	{attribute 'TcIecLibraryType'}
	{attribute 'external_name' := 'F_VN_ReadDataMatrixCode_GUID_2844DFEA_73D9_3166_383A_C70A652858C4'}
	(* Detect and interpret a data matrix code within the provided image. *)
	FUNCTION F_VN_ReadDataMatrixCode : HRESULT
	VAR_INPUT
		ipSrcImage	:	ITcVnImage;	(* Source image (USINT elements, 1 or 3 channels) *)
		ipDecodedData	:	REFERENCE TO ITcVnContainer;	(* Returns the decoded code (ContainerType_Vector_String_SINT) *)
		hrPrev	:	HRESULT;	(* HRESULT indicating the result of previous operations (If SUCCEEDED(hrPrev) equals false, no operation is executed.) *)
	END_VAR

END_FUNCTION

// Functions/Code Reading/F_VN_ReadDataMatrixCodeExp

	{attribute 'TcIecLibraryType'}
	{attribute 'external_name' := 'F_VN_ReadDataMatrixCodeExp_GUID_B61F2F2C_5B12_3E0F_1052_05187753987C'}
	(* Detect and interpret a data matrix code within the provided image. *)
	FUNCTION F_VN_ReadDataMatrixCodeExp : HRESULT
	VAR_INPUT
		ipSrcImage	:	ITcVnImage;	(* Source image (USINT elements, 1 or 3 channels) *)
		ipDecodedData	:	REFERENCE TO ITcVnContainer;	(* Returns the decoded code (ContainerType_Vector_String_SINT) *)
		ipContours	:	REFERENCE TO ITcVnContainer;	(* Returns the code positions as contours (ContainerType_Vector_Vector_TcVnPoint2_DINT) *)
		nCodeNumber	:	DINT;	(* Number of data matrix codes that should be detected within the provided image. (If set to -1, it is tried to detect all data matrix codes.) *)
		eSearchStrategy	:	UDINT;	(* Used search strategy (ETcVn2dCodeSearchStrategy) *)
		hrPrev	:	HRESULT;	(* HRESULT indicating the result of previous operations (If SUCCEEDED(hrPrev) equals false, no operation is executed.) *)
	END_VAR

END_FUNCTION

// Functions/Code Reading/F_VN_ReadPharmaCode

	{attribute 'TcIecLibraryType'}
	{attribute 'external_name' := 'F_VN_ReadPharmaCode_GUID_7AF29CDE_1633_3CD4_1E1F_1FA9D1B23190'}
	(* Detect and interpret a pharma code within the provided image.
				Can be canceled by Watchdog. *)
	FUNCTION F_VN_ReadPharmaCode : HRESULT
	VAR_INPUT
		ipSrcImage	:	ITcVnImage;	(* Source image (1 channel (all element types) or 3 channel with elements of type TCVN_ET_USINT, TCVN_ET_UINT or TCVN_ET_REAL (3 channel input is expected to be RGB and internally converted to Gray)) *)
		ipDecodedData	:	REFERENCE TO ITcVnContainer;	(* Returns the decoded code (ContainerType_Vector_String_SINT) *)
		hrPrev	:	HRESULT;	(* HRESULT indicating the result of previous operations (If SUCCEEDED(hrPrev) equals false, no operation is executed.) *)
	END_VAR

END_FUNCTION

// Functions/Code Reading/F_VN_ReadPharmaCodeExp

	{attribute 'TcIecLibraryType'}
	{attribute 'external_name' := 'F_VN_ReadPharmaCodeExp_GUID_7FECB9FD_CF47_3BD7_11A2_73B8C61437DB'}
	(* Detect and interpret a pharma code within the provided image.
				Can be canceled by Watchdog. *)
	FUNCTION F_VN_ReadPharmaCodeExp : HRESULT
	VAR_INPUT
		ipSrcImage	:	ITcVnImage;	(* Source image (1 channel (all element types) or 3 channel with elements of type TCVN_ET_USINT, TCVN_ET_UINT or TCVN_ET_REAL (3 channel input is expected to be RGB and internally converted to Gray)) *)
		ipDecodedData	:	REFERENCE TO ITcVnContainer;	(* Returns the decoded code (ContainerType_Vector_String_SINT) *)
		ipContours	:	REFERENCE TO ITcVnContainer;	(* Returns the code positions as contours (ContainerType_Vector_Vector_TcVnPoint2_DINT) *)
		nCodeNumber	:	DINT;	(* Number of pharma codes that should be detected within the provided image (currently only 1 supported). *)
		nMinBarNumber	:	INT;	(* Minimal number of (dark) bars that codes must have. *)
		hrPrev	:	HRESULT;	(* HRESULT indicating the result of previous operations (If SUCCEEDED(hrPrev) equals false, no operation is executed.) *)
	END_VAR

END_FUNCTION

// Functions/Code Reading/F_VN_ReadQRCode

	{attribute 'TcIecLibraryType'}
	{attribute 'external_name' := 'F_VN_ReadQRCode_GUID_FDADFE2B_041B_3714_35C5_CCC4D2EB5C52'}
	(* Detect and interpret a QR code within the provided image.
          Can be canceled by Watchdog. *)
	FUNCTION F_VN_ReadQRCode : HRESULT
	VAR_INPUT
		ipSrcImage	:	ITcVnImage;	(* Source image (USINT elements, 1 channel or 3 channel (3 channel input is expected to be RGB and internally converted to Gray)) *)
		ipDecodedData	:	REFERENCE TO ITcVnContainer;	(* Returns the decoded code (ContainerType_Vector_String_SINT) *)
		hrPrev	:	HRESULT;	(* HRESULT indicating the result of previous operations (If SUCCEEDED(hrPrev) equals false, no operation is executed.) *)
	END_VAR

END_FUNCTION

// Functions/Code Reading/F_VN_ReadQRCodeExp

	{attribute 'TcIecLibraryType'}
	{attribute 'external_name' := 'F_VN_ReadQRCodeExp_GUID_701D058E_193D_312D_3EA8_971256078500'}
	(* Detect and interpret a QR code within the provided image.
          Can be canceled by Watchdog. *)
	FUNCTION F_VN_ReadQRCodeExp : HRESULT
	VAR_INPUT
		ipSrcImage	:	ITcVnImage;	(* Source image (USINT elements, 1 channel or 3 channel (3 channel input is expected to be RGB and internally converted to Gray)) *)
		ipDecodedData	:	REFERENCE TO ITcVnContainer;	(* Returns the decoded code (ContainerType_Vector_String_SINT) *)
		ipContours	:	REFERENCE TO ITcVnContainer;	(* Returns the code positions as contours (ContainerType_Vector_Vector_TcVnPoint2_DINT) *)
		nCodeNumber	:	DINT;	(* Number of QR codes that should be detected within the provided image (currently only 1 supported). *)
		eSearchStrategy	:	UDINT;	(* Used search strategy (ETcVn2dCodeSearchStrategy) *)
		hrPrev	:	HRESULT;	(* HRESULT indicating the result of previous operations (If SUCCEEDED(hrPrev) equals false, no operation is executed.) *)
	END_VAR

END_FUNCTION

// Functions/Algebraic Container Operations/F_VN_AddToContainerElements/F_VN_AddToContainerElements_DINT

	{attribute 'TcIecLibraryType'}
	{attribute 'external_name' := 'F_VN_AddToContainerElements_DINT_GUID_5B932B1D_0AB0_3885_2F50_15772C7465B6'}
	(* Add a value to each container element. *)
	FUNCTION F_VN_AddToContainerElements_DINT : HRESULT
	VAR_INPUT
		nValue	:	DINT;	(* Value *)
		ipContainer	:	ITcVnContainer;	(* Container with DINT elements *)
		hrPrev	:	HRESULT;	(* HRESULT indicating the result of previous operations (If SUCCEEDED(hrPrev) equals false, no operation is executed.) *)
	END_VAR

END_FUNCTION

// Functions/Algebraic Container Operations/F_VN_AddToContainerElements/F_VN_AddToContainerElements_INT

	{attribute 'TcIecLibraryType'}
	{attribute 'external_name' := 'F_VN_AddToContainerElements_INT_GUID_8666D2A8_02E9_3A45_051D_A4854190DF10'}
	(* Add a value to each container element. *)
	FUNCTION F_VN_AddToContainerElements_INT : HRESULT
	VAR_INPUT
		nValue	:	INT;	(* Value *)
		ipContainer	:	ITcVnContainer;	(* Container with INT elements *)
		hrPrev	:	HRESULT;	(* HRESULT indicating the result of previous operations (If SUCCEEDED(hrPrev) equals false, no operation is executed.) *)
	END_VAR

END_FUNCTION

// Functions/Algebraic Container Operations/F_VN_AddToContainerElements/F_VN_AddToContainerElements_LREAL

	{attribute 'TcIecLibraryType'}
	{attribute 'external_name' := 'F_VN_AddToContainerElements_LREAL_GUID_E41AE159_0A04_3EFE_16AB_C8BFD4EDC43A'}
	(* Add a value to each container element. *)
	FUNCTION F_VN_AddToContainerElements_LREAL : HRESULT
	VAR_INPUT
		fValue	:	LREAL;	(* Value *)
		ipContainer	:	ITcVnContainer;	(* Container with LREAL elements *)
		hrPrev	:	HRESULT;	(* HRESULT indicating the result of previous operations (If SUCCEEDED(hrPrev) equals false, no operation is executed.) *)
	END_VAR

END_FUNCTION

// Functions/Algebraic Container Operations/F_VN_AddToContainerElements/F_VN_AddToContainerElements_REAL

	{attribute 'TcIecLibraryType'}
	{attribute 'external_name' := 'F_VN_AddToContainerElements_REAL_GUID_692D4EAD_61C5_34E3_07CE_2D6EFBC619FC'}
	(* Add a value to each container element. *)
	FUNCTION F_VN_AddToContainerElements_REAL : HRESULT
	VAR_INPUT
		fValue	:	REAL;	(* Value *)
		ipContainer	:	ITcVnContainer;	(* Container with REAL elements *)
		hrPrev	:	HRESULT;	(* HRESULT indicating the result of previous operations (If SUCCEEDED(hrPrev) equals false, no operation is executed.) *)
	END_VAR

END_FUNCTION

// Functions/Algebraic Container Operations/F_VN_AddToContainerElements/F_VN_AddToContainerElements_SINT

	{attribute 'TcIecLibraryType'}
	{attribute 'external_name' := 'F_VN_AddToContainerElements_SINT_GUID_226FCB6F_5B19_30F7_05FC_4AEA7FD84914'}
	(* Add a value to each container element. *)
	FUNCTION F_VN_AddToContainerElements_SINT : HRESULT
	VAR_INPUT
		nValue	:	SINT;	(* Value *)
		ipContainer	:	ITcVnContainer;	(* Container with SINT elements *)
		hrPrev	:	HRESULT;	(* HRESULT indicating the result of previous operations (If SUCCEEDED(hrPrev) equals false, no operation is executed.) *)
	END_VAR

END_FUNCTION

// Functions/Algebraic Container Operations/F_VN_AddToContainerElements/F_VN_AddToContainerElements_TcVnKeyPoint

	{attribute 'TcIecLibraryType'}
	{attribute 'external_name' := 'F_VN_AddToContainerElements_TcVnKeyPoint_GUID_3B5F4B12_691D_304E_2813_D0B80607BE3C'}
	(* Add a value to each container element. *)
	FUNCTION F_VN_AddToContainerElements_TcVnKeyPoint : HRESULT
	VAR_INPUT
		stValue	:	REFERENCE TO TcVnKeyPoint;	(* Value *)
		ipContainer	:	ITcVnContainer;	(* Container with TcVnKeyPoint elements *)
		hrPrev	:	HRESULT;	(* HRESULT indicating the result of previous operations (If SUCCEEDED(hrPrev) equals false, no operation is executed.) *)
	END_VAR

END_FUNCTION

// Functions/Algebraic Container Operations/F_VN_AddToContainerElements/F_VN_AddToContainerElements_TcVnPoint2_DINT

	{attribute 'TcIecLibraryType'}
	{attribute 'external_name' := 'F_VN_AddToContainerElements_TcVnPoint2_DINT_GUID_01834351_EA53_3313_1ABA_CB9AAEF6914A'}
	(* Add a value to each container element. *)
	FUNCTION F_VN_AddToContainerElements_TcVnPoint2_DINT : HRESULT
	VAR_INPUT
		aValue	:	REFERENCE TO TcVnPoint2_DINT;	(* Value *)
		ipContainer	:	ITcVnContainer;	(* Container with TcVnPoint2_DINT elements *)
		hrPrev	:	HRESULT;	(* HRESULT indicating the result of previous operations (If SUCCEEDED(hrPrev) equals false, no operation is executed.) *)
	END_VAR

END_FUNCTION

// Functions/Algebraic Container Operations/F_VN_AddToContainerElements/F_VN_AddToContainerElements_TcVnPoint2_LREAL

	{attribute 'TcIecLibraryType'}
	{attribute 'external_name' := 'F_VN_AddToContainerElements_TcVnPoint2_LREAL_GUID_43701B1D_E3A8_30C8_24E6_54A2EFDCAA91'}
	(* Add a value to each container element. *)
	FUNCTION F_VN_AddToContainerElements_TcVnPoint2_LREAL : HRESULT
	VAR_INPUT
		aValue	:	REFERENCE TO TcVnPoint2_LREAL;	(* Value *)
		ipContainer	:	ITcVnContainer;	(* Container with TcVnPoint2_LREAL elements *)
		hrPrev	:	HRESULT;	(* HRESULT indicating the result of previous operations (If SUCCEEDED(hrPrev) equals false, no operation is executed.) *)
	END_VAR

END_FUNCTION

// Functions/Algebraic Container Operations/F_VN_AddToContainerElements/F_VN_AddToContainerElements_TcVnPoint2_REAL

	{attribute 'TcIecLibraryType'}
	{attribute 'external_name' := 'F_VN_AddToContainerElements_TcVnPoint2_REAL_GUID_00905747_5375_3335_13FD_44D74374D245'}
	(* Add a value to each container element. *)
	FUNCTION F_VN_AddToContainerElements_TcVnPoint2_REAL : HRESULT
	VAR_INPUT
		aValue	:	REFERENCE TO TcVnPoint2_REAL;	(* Value *)
		ipContainer	:	ITcVnContainer;	(* Container with TcVnPoint2_REAL elements *)
		hrPrev	:	HRESULT;	(* HRESULT indicating the result of previous operations (If SUCCEEDED(hrPrev) equals false, no operation is executed.) *)
	END_VAR

END_FUNCTION

// Functions/Algebraic Container Operations/F_VN_AddToContainerElements/F_VN_AddToContainerElements_TcVnPoint3_LREAL

	{attribute 'TcIecLibraryType'}
	{attribute 'external_name' := 'F_VN_AddToContainerElements_TcVnPoint3_LREAL_GUID_839DAD36_31CD_3F38_311A_A016EB995C42'}
	(* Add a value to each container element. *)
	FUNCTION F_VN_AddToContainerElements_TcVnPoint3_LREAL : HRESULT
	VAR_INPUT
		aValue	:	REFERENCE TO TcVnPoint3_LREAL;	(* Value *)
		ipContainer	:	ITcVnContainer;	(* Container with TcVnPoint3_LREAL elements *)
		hrPrev	:	HRESULT;	(* HRESULT indicating the result of previous operations (If SUCCEEDED(hrPrev) equals false, no operation is executed.) *)
	END_VAR

END_FUNCTION

// Functions/Algebraic Container Operations/F_VN_AddToContainerElements/F_VN_AddToContainerElements_TcVnPoint3_REAL

	{attribute 'TcIecLibraryType'}
	{attribute 'external_name' := 'F_VN_AddToContainerElements_TcVnPoint3_REAL_GUID_7F806659_1D47_3D35_077C_CC3B8A9E940F'}
	(* Add a value to each container element. *)
	FUNCTION F_VN_AddToContainerElements_TcVnPoint3_REAL : HRESULT
	VAR_INPUT
		aValue	:	REFERENCE TO TcVnPoint3_REAL;	(* Value *)
		ipContainer	:	ITcVnContainer;	(* Container with TcVnPoint3_REAL elements *)
		hrPrev	:	HRESULT;	(* HRESULT indicating the result of previous operations (If SUCCEEDED(hrPrev) equals false, no operation is executed.) *)
	END_VAR

END_FUNCTION

// Functions/Algebraic Container Operations/F_VN_AddToContainerElements/F_VN_AddToContainerElements_TcVnRectangle_DINT

	{attribute 'TcIecLibraryType'}
	{attribute 'external_name' := 'F_VN_AddToContainerElements_TcVnRectangle_DINT_GUID_5752E0A5_0126_3CCC_0ED6_0FAF696F41AB'}
	(* Add a value to each container element. *)
	FUNCTION F_VN_AddToContainerElements_TcVnRectangle_DINT : HRESULT
	VAR_INPUT
		stValue	:	REFERENCE TO TcVnRectangle_DINT;	(* Value *)
		ipContainer	:	ITcVnContainer;	(* Container with TcVnRectangle_DINT elements *)
		hrPrev	:	HRESULT;	(* HRESULT indicating the result of previous operations (If SUCCEEDED(hrPrev) equals false, no operation is executed.) *)
	END_VAR

END_FUNCTION

// Functions/Algebraic Container Operations/F_VN_AddToContainerElements/F_VN_AddToContainerElements_TcVnVector2_DINT

	{attribute 'TcIecLibraryType'}
	{attribute 'external_name' := 'F_VN_AddToContainerElements_TcVnVector2_DINT_GUID_FD05239B_FA44_389E_2792_06A9AFDB811F'}
	(* Add a value to each container element. *)
	FUNCTION F_VN_AddToContainerElements_TcVnVector2_DINT : HRESULT
	VAR_INPUT
		aValue	:	REFERENCE TO TcVnVector2_DINT;	(* Value *)
		ipContainer	:	ITcVnContainer;	(* Container with TcVnVector2_DINT elements *)
		hrPrev	:	HRESULT;	(* HRESULT indicating the result of previous operations (If SUCCEEDED(hrPrev) equals false, no operation is executed.) *)
	END_VAR

END_FUNCTION

// Functions/Algebraic Container Operations/F_VN_AddToContainerElements/F_VN_AddToContainerElements_TcVnVector2_INT

	{attribute 'TcIecLibraryType'}
	{attribute 'external_name' := 'F_VN_AddToContainerElements_TcVnVector2_INT_GUID_5A7959AB_7E96_36FB_0F59_3CCB450F9AC2'}
	(* Add a value to each container element. *)
	FUNCTION F_VN_AddToContainerElements_TcVnVector2_INT : HRESULT
	VAR_INPUT
		aValue	:	REFERENCE TO TcVnVector2_INT;	(* Value *)
		ipContainer	:	ITcVnContainer;	(* Container with TcVnVector2_INT elements *)
		hrPrev	:	HRESULT;	(* HRESULT indicating the result of previous operations (If SUCCEEDED(hrPrev) equals false, no operation is executed.) *)
	END_VAR

END_FUNCTION

// Functions/Algebraic Container Operations/F_VN_AddToContainerElements/F_VN_AddToContainerElements_TcVnVector2_REAL

	{attribute 'TcIecLibraryType'}
	{attribute 'external_name' := 'F_VN_AddToContainerElements_TcVnVector2_REAL_GUID_1870524F_E8DF_343A_1F0A_A50A67E87D79'}
	(* Add a value to each container element. *)
	FUNCTION F_VN_AddToContainerElements_TcVnVector2_REAL : HRESULT
	VAR_INPUT
		aValue	:	REFERENCE TO TcVnVector2_REAL;	(* Value *)
		ipContainer	:	ITcVnContainer;	(* Container with TcVnVector2_REAL elements *)
		hrPrev	:	HRESULT;	(* HRESULT indicating the result of previous operations (If SUCCEEDED(hrPrev) equals false, no operation is executed.) *)
	END_VAR

END_FUNCTION

// Functions/Algebraic Container Operations/F_VN_AddToContainerElements/F_VN_AddToContainerElements_TcVnVector2_SINT

	{attribute 'TcIecLibraryType'}
	{attribute 'external_name' := 'F_VN_AddToContainerElements_TcVnVector2_SINT_GUID_BA86B28B_BD11_3A77_358B_D5CC18E5F5D5'}
	(* Add a value to each container element. *)
	FUNCTION F_VN_AddToContainerElements_TcVnVector2_SINT : HRESULT
	VAR_INPUT
		aValue	:	REFERENCE TO TcVnVector2_SINT;	(* Value *)
		ipContainer	:	ITcVnContainer;	(* Container with TcVnVector2_SINT elements *)
		hrPrev	:	HRESULT;	(* HRESULT indicating the result of previous operations (If SUCCEEDED(hrPrev) equals false, no operation is executed.) *)
	END_VAR

END_FUNCTION

// Functions/Algebraic Container Operations/F_VN_AddToContainerElements/F_VN_AddToContainerElements_TcVnVector2_UINT

	{attribute 'TcIecLibraryType'}
	{attribute 'external_name' := 'F_VN_AddToContainerElements_TcVnVector2_UINT_GUID_56354970_50D0_3E9A_1D26_63220324D232'}
	(* Add a value to each container element. *)
	FUNCTION F_VN_AddToContainerElements_TcVnVector2_UINT : HRESULT
	VAR_INPUT
		aValue	:	REFERENCE TO TcVnVector2_UINT;	(* Value *)
		ipContainer	:	ITcVnContainer;	(* Container with TcVnVector2_UINT elements *)
		hrPrev	:	HRESULT;	(* HRESULT indicating the result of previous operations (If SUCCEEDED(hrPrev) equals false, no operation is executed.) *)
	END_VAR

END_FUNCTION

// Functions/Algebraic Container Operations/F_VN_AddToContainerElements/F_VN_AddToContainerElements_TcVnVector2_USINT

	{attribute 'TcIecLibraryType'}
	{attribute 'external_name' := 'F_VN_AddToContainerElements_TcVnVector2_USINT_GUID_19808A36_72A8_3C12_006D_40846B9F72C1'}
	(* Add a value to each container element. *)
	FUNCTION F_VN_AddToContainerElements_TcVnVector2_USINT : HRESULT
	VAR_INPUT
		aValue	:	REFERENCE TO TcVnVector2_USINT;	(* Value *)
		ipContainer	:	ITcVnContainer;	(* Container with TcVnVector2_USINT elements *)
		hrPrev	:	HRESULT;	(* HRESULT indicating the result of previous operations (If SUCCEEDED(hrPrev) equals false, no operation is executed.) *)
	END_VAR

END_FUNCTION

// Functions/Algebraic Container Operations/F_VN_AddToContainerElements/F_VN_AddToContainerElements_TcVnVector3_INT

	{attribute 'TcIecLibraryType'}
	{attribute 'external_name' := 'F_VN_AddToContainerElements_TcVnVector3_INT_GUID_71DC03E7_7327_3F01_0329_49D058A39A31'}
	(* Add a value to each container element. *)
	FUNCTION F_VN_AddToContainerElements_TcVnVector3_INT : HRESULT
	VAR_INPUT
		aValue	:	REFERENCE TO TcVnVector3_INT;	(* Value *)
		ipContainer	:	ITcVnContainer;	(* Container with TcVnVector3_INT elements *)
		hrPrev	:	HRESULT;	(* HRESULT indicating the result of previous operations (If SUCCEEDED(hrPrev) equals false, no operation is executed.) *)
	END_VAR

END_FUNCTION

// Functions/Algebraic Container Operations/F_VN_AddToContainerElements/F_VN_AddToContainerElements_TcVnVector3_REAL

	{attribute 'TcIecLibraryType'}
	{attribute 'external_name' := 'F_VN_AddToContainerElements_TcVnVector3_REAL_GUID_07AE301A_FCD1_34F3_164A_C1B5204DF30F'}
	(* Add a value to each container element. *)
	FUNCTION F_VN_AddToContainerElements_TcVnVector3_REAL : HRESULT
	VAR_INPUT
		aValue	:	REFERENCE TO TcVnVector3_REAL;	(* Value *)
		ipContainer	:	ITcVnContainer;	(* Container with TcVnVector3_REAL elements *)
		hrPrev	:	HRESULT;	(* HRESULT indicating the result of previous operations (If SUCCEEDED(hrPrev) equals false, no operation is executed.) *)
	END_VAR

END_FUNCTION

// Functions/Algebraic Container Operations/F_VN_AddToContainerElements/F_VN_AddToContainerElements_TcVnVector3_SINT

	{attribute 'TcIecLibraryType'}
	{attribute 'external_name' := 'F_VN_AddToContainerElements_TcVnVector3_SINT_GUID_6B5F8825_61DA_34E0_2CA0_F82329D5E791'}
	(* Add a value to each container element. *)
	FUNCTION F_VN_AddToContainerElements_TcVnVector3_SINT : HRESULT
	VAR_INPUT
		aValue	:	REFERENCE TO TcVnVector3_SINT;	(* Value *)
		ipContainer	:	ITcVnContainer;	(* Container with TcVnVector3_SINT elements *)
		hrPrev	:	HRESULT;	(* HRESULT indicating the result of previous operations (If SUCCEEDED(hrPrev) equals false, no operation is executed.) *)
	END_VAR

END_FUNCTION

// Functions/Algebraic Container Operations/F_VN_AddToContainerElements/F_VN_AddToContainerElements_TcVnVector3_UINT

	{attribute 'TcIecLibraryType'}
	{attribute 'external_name' := 'F_VN_AddToContainerElements_TcVnVector3_UINT_GUID_C23A5AA0_44F7_3E02_1B8F_AF04E59BD1A4'}
	(* Add a value to each container element. *)
	FUNCTION F_VN_AddToContainerElements_TcVnVector3_UINT : HRESULT
	VAR_INPUT
		aValue	:	REFERENCE TO TcVnVector3_UINT;	(* Value *)
		ipContainer	:	ITcVnContainer;	(* Container with TcVnVector3_UINT elements *)
		hrPrev	:	HRESULT;	(* HRESULT indicating the result of previous operations (If SUCCEEDED(hrPrev) equals false, no operation is executed.) *)
	END_VAR

END_FUNCTION

// Functions/Algebraic Container Operations/F_VN_AddToContainerElements/F_VN_AddToContainerElements_TcVnVector3_USINT

	{attribute 'TcIecLibraryType'}
	{attribute 'external_name' := 'F_VN_AddToContainerElements_TcVnVector3_USINT_GUID_D752658B_8056_3256_1C1B_709D22CABB66'}
	(* Add a value to each container element. *)
	FUNCTION F_VN_AddToContainerElements_TcVnVector3_USINT : HRESULT
	VAR_INPUT
		aValue	:	REFERENCE TO TcVnVector3_USINT;	(* Value *)
		ipContainer	:	ITcVnContainer;	(* Container with TcVnVector3_USINT elements *)
		hrPrev	:	HRESULT;	(* HRESULT indicating the result of previous operations (If SUCCEEDED(hrPrev) equals false, no operation is executed.) *)
	END_VAR

END_FUNCTION

// Functions/Algebraic Container Operations/F_VN_AddToContainerElements/F_VN_AddToContainerElements_TcVnVector4_DINT

	{attribute 'TcIecLibraryType'}
	{attribute 'external_name' := 'F_VN_AddToContainerElements_TcVnVector4_DINT_GUID_D742BE97_80DB_3CB5_027E_781E374D608F'}
	(* Add a value to each container element. *)
	FUNCTION F_VN_AddToContainerElements_TcVnVector4_DINT : HRESULT
	VAR_INPUT
		aValue	:	REFERENCE TO TcVnVector4_DINT;	(* Value *)
		ipContainer	:	ITcVnContainer;	(* Container with TcVnVector4_DINT elements *)
		hrPrev	:	HRESULT;	(* HRESULT indicating the result of previous operations (If SUCCEEDED(hrPrev) equals false, no operation is executed.) *)
	END_VAR

END_FUNCTION

// Functions/Algebraic Container Operations/F_VN_AddToContainerElements/F_VN_AddToContainerElements_TcVnVector4_INT

	{attribute 'TcIecLibraryType'}
	{attribute 'external_name' := 'F_VN_AddToContainerElements_TcVnVector4_INT_GUID_57836443_D91C_30AD_0584_7CCF6B06E1D4'}
	(* Add a value to each container element. *)
	FUNCTION F_VN_AddToContainerElements_TcVnVector4_INT : HRESULT
	VAR_INPUT
		aValue	:	REFERENCE TO TcVnVector4_INT;	(* Value *)
		ipContainer	:	ITcVnContainer;	(* Container with TcVnVector4_INT elements *)
		hrPrev	:	HRESULT;	(* HRESULT indicating the result of previous operations (If SUCCEEDED(hrPrev) equals false, no operation is executed.) *)
	END_VAR

END_FUNCTION

// Functions/Algebraic Container Operations/F_VN_AddToContainerElements/F_VN_AddToContainerElements_TcVnVector4_LREAL

	{attribute 'TcIecLibraryType'}
	{attribute 'external_name' := 'F_VN_AddToContainerElements_TcVnVector4_LREAL_GUID_360561FB_FBFC_3471_3F24_900DC5ABA6EC'}
	(* Add a value to each container element. *)
	FUNCTION F_VN_AddToContainerElements_TcVnVector4_LREAL : HRESULT
	VAR_INPUT
		aValue	:	REFERENCE TO TcVnVector4_LREAL;	(* Value *)
		ipContainer	:	ITcVnContainer;	(* Container with TcVnVector4_LREAL elements *)
		hrPrev	:	HRESULT;	(* HRESULT indicating the result of previous operations (If SUCCEEDED(hrPrev) equals false, no operation is executed.) *)
	END_VAR

END_FUNCTION

// Functions/Algebraic Container Operations/F_VN_AddToContainerElements/F_VN_AddToContainerElements_TcVnVector4_SINT

	{attribute 'TcIecLibraryType'}
	{attribute 'external_name' := 'F_VN_AddToContainerElements_TcVnVector4_SINT_GUID_1820B1AC_0FF9_3EE1_38CE_685FDE758958'}
	(* Add a value to each container element. *)
	FUNCTION F_VN_AddToContainerElements_TcVnVector4_SINT : HRESULT
	VAR_INPUT
		aValue	:	REFERENCE TO TcVnVector4_SINT;	(* Value *)
		ipContainer	:	ITcVnContainer;	(* Container with TcVnVector4_SINT elements *)
		hrPrev	:	HRESULT;	(* HRESULT indicating the result of previous operations (If SUCCEEDED(hrPrev) equals false, no operation is executed.) *)
	END_VAR

END_FUNCTION

// Functions/Algebraic Container Operations/F_VN_AddToContainerElements/F_VN_AddToContainerElements_TcVnVector4_UINT

	{attribute 'TcIecLibraryType'}
	{attribute 'external_name' := 'F_VN_AddToContainerElements_TcVnVector4_UINT_GUID_5187AFB3_19BE_3EE8_32AD_0FFCFCC25933'}
	(* Add a value to each container element. *)
	FUNCTION F_VN_AddToContainerElements_TcVnVector4_UINT : HRESULT
	VAR_INPUT
		aValue	:	REFERENCE TO TcVnVector4_UINT;	(* Value *)
		ipContainer	:	ITcVnContainer;	(* Container with TcVnVector4_UINT elements *)
		hrPrev	:	HRESULT;	(* HRESULT indicating the result of previous operations (If SUCCEEDED(hrPrev) equals false, no operation is executed.) *)
	END_VAR

END_FUNCTION

// Functions/Algebraic Container Operations/F_VN_AddToContainerElements/F_VN_AddToContainerElements_TcVnVector4_USINT

	{attribute 'TcIecLibraryType'}
	{attribute 'external_name' := 'F_VN_AddToContainerElements_TcVnVector4_USINT_GUID_77580D86_B358_375A_06A3_8BDBEA39CE74'}
	(* Add a value to each container element. *)
	FUNCTION F_VN_AddToContainerElements_TcVnVector4_USINT : HRESULT
	VAR_INPUT
		aValue	:	REFERENCE TO TcVnVector4_USINT;	(* Value *)
		ipContainer	:	ITcVnContainer;	(* Container with TcVnVector4_USINT elements *)
		hrPrev	:	HRESULT;	(* HRESULT indicating the result of previous operations (If SUCCEEDED(hrPrev) equals false, no operation is executed.) *)
	END_VAR

END_FUNCTION

// Functions/Algebraic Container Operations/F_VN_AddToContainerElements/F_VN_AddToContainerElements_UDINT

	{attribute 'TcIecLibraryType'}
	{attribute 'external_name' := 'F_VN_AddToContainerElements_UDINT_GUID_5ECD52C6_7D8F_3D13_28F8_D2F1CCB21427'}
	(* Add a value to each container element. *)
	FUNCTION F_VN_AddToContainerElements_UDINT : HRESULT
	VAR_INPUT
		nValue	:	UDINT;	(* Value *)
		ipContainer	:	ITcVnContainer;	(* Container with UDINT elements *)
		hrPrev	:	HRESULT;	(* HRESULT indicating the result of previous operations (If SUCCEEDED(hrPrev) equals false, no operation is executed.) *)
	END_VAR

END_FUNCTION

// Functions/Algebraic Container Operations/F_VN_AddToContainerElements/F_VN_AddToContainerElements_UINT

	{attribute 'TcIecLibraryType'}
	{attribute 'external_name' := 'F_VN_AddToContainerElements_UINT_GUID_AAC9CFC5_57F2_382F_1BD9_9DFEB6B09CFB'}
	(* Add a value to each container element. *)
	FUNCTION F_VN_AddToContainerElements_UINT : HRESULT
	VAR_INPUT
		nValue	:	UINT;	(* Value *)
		ipContainer	:	ITcVnContainer;	(* Container with UINT elements *)
		hrPrev	:	HRESULT;	(* HRESULT indicating the result of previous operations (If SUCCEEDED(hrPrev) equals false, no operation is executed.) *)
	END_VAR

END_FUNCTION

// Functions/Algebraic Container Operations/F_VN_AddToContainerElements/F_VN_AddToContainerElements_ULINT

	{attribute 'TcIecLibraryType'}
	{attribute 'external_name' := 'F_VN_AddToContainerElements_ULINT_GUID_85BFEBDA_E705_31D3_2B59_BA00C1290486'}
	(* Add a value to each container element. *)
	FUNCTION F_VN_AddToContainerElements_ULINT : HRESULT
	VAR_INPUT
		nValue	:	ULINT;	(* Value *)
		ipContainer	:	ITcVnContainer;	(* Container with ULINT elements *)
		hrPrev	:	HRESULT;	(* HRESULT indicating the result of previous operations (If SUCCEEDED(hrPrev) equals false, no operation is executed.) *)
	END_VAR

END_FUNCTION

// Functions/Algebraic Container Operations/F_VN_AddToContainerElements/F_VN_AddToContainerElements_USINT

	{attribute 'TcIecLibraryType'}
	{attribute 'external_name' := 'F_VN_AddToContainerElements_USINT_GUID_5BF3EAE4_887F_3F25_01F9_F187751B7D61'}
	(* Add a value to each container element. *)
	FUNCTION F_VN_AddToContainerElements_USINT : HRESULT
	VAR_INPUT
		nValue	:	USINT;	(* Value *)
		ipContainer	:	ITcVnContainer;	(* Container with USINT elements *)
		hrPrev	:	HRESULT;	(* HRESULT indicating the result of previous operations (If SUCCEEDED(hrPrev) equals false, no operation is executed.) *)
	END_VAR

END_FUNCTION

// Functions/Image Analysis/Object Detection/F_VN_AdjustActiveContour

	{attribute 'TcIecLibraryType'}
	{attribute 'external_name' := 'F_VN_AdjustActiveContour_GUID_E8A83B8A_FFAF_376E_0EAC_1914E2C30A5B'}
	(* Adjust active contour (snake) in order to minimize its cummulative (internal and external) energy. *)
	FUNCTION F_VN_AdjustActiveContour : HRESULT
	VAR_INPUT
		ipImage	:	ITcVnImage;	(* Source image (1 channel, USINT elements) *)
		ipActiveContour	:	ITcVnContainer;	(* Initial contour, which will be adjusted *)
		fAlpha	:	REAL;	(* Continuity energy coefficient *)
		fBeta	:	REAL;	(* Curvature energy coefficient *)
		fGamma	:	REAL;	(* Image energy coefficient *)
		nWindowWidth	:	UDINT;	(* Windows width (3, 5, 7, ...) *)
		nWindowHeight	:	UDINT;	(* Windows height (3, 5, 7, ...) *)
		nMaxIterations	:	UDINT;	(* Maximum iterations *)
		bUseGradient	:	BOOL;	(* If true, the gradient magnitude is used as image energy (otherwise: pixel intensity) *)
		hrPrev	:	HRESULT;	(* HRESULT indicating the result of previous operations (If SUCCEEDED(hrPrev) equals false, no operation is executed.) *)
	END_VAR

END_FUNCTION

// Functions/Image Analysis/Object Detection/F_VN_DetectBlobs

	{attribute 'TcIecLibraryType'}
	{attribute 'external_name' := 'F_VN_DetectBlobs_GUID_D96B8C6D_95DC_37E7_33AE_CFA61E2C6332'}
	(* Detects blob-contours. Applies a threshold, a contour search and offers several options for filtering the found contours. Provides easy setup for multiple thresholds and combination of results. *)
	FUNCTION F_VN_DetectBlobs : HRESULT
	VAR_INPUT
		ipSrcImage	:	ITcVnImage;	(* Source image (USINT or REAL, 1 channel or 3 channel (3 channel input is expected to be RGB and internally converted to Gray)) *)
		ipBlobContours	:	REFERENCE TO ITcVnContainer;	(* Returns a container which is filled with the found contours (ContainerType_Vector_Vector_TcVnPoint2_DINT; The elements of this container are single contours. Non-zero interface pointers are reused.) *)
		stParams	:	REFERENCE TO TcVnParamsBlobDetection;	(* Parameters to filter the detected contours. *)
		hrPrev	:	HRESULT;	(* HRESULT indicating the result of previous operations (If SUCCEEDED(hrPrev) equals false, no operation is executed.) *)
	END_VAR

END_FUNCTION

// Functions/Image Analysis/Object Detection/F_VN_DetectBlobsExp

	{attribute 'TcIecLibraryType'}
	{attribute 'external_name' := 'F_VN_DetectBlobsExp_GUID_FC112C44_43B7_3777_1919_1F0811271198'}
	(* Detects blob-contours. Applies a threshold, a contour search and offers several options for filtering the found contours. Provides easy setup for multiple thresholds and combination of results. (expert function) *)
	FUNCTION F_VN_DetectBlobsExp : HRESULT
	VAR_INPUT
		ipSrcImage	:	ITcVnImage;	(* Source image (USINT or REAL, 1 channel or 3 channel (3 channel input is expected to be RGB and internally converted to Gray)) *)
		ipBlobContours	:	REFERENCE TO ITcVnContainer;	(* Returns a container which is filled with the found contours (ContainerType_Vector_Vector_TcVnPoint2_DINT; The elements of this container are single contours. Non-zero interface pointers are reused.) *)
		stParams	:	REFERENCE TO TcVnParamsBlobDetection;	(* Parameters to filter the detected contours. *)
		aOffset	:	REFERENCE TO TcVnPoint;	(* Offset by which every contour point is shifted *)
		hrPrev	:	HRESULT;	(* HRESULT indicating the result of previous operations (If SUCCEEDED(hrPrev) equals false, no operation is executed.) *)
	END_VAR

END_FUNCTION

// Functions/Image Analysis/Object Detection/F_VN_FindContourHierarchyExp

	{attribute 'TcIecLibraryType'}
	{attribute 'external_name' := 'F_VN_FindContourHierarchyExp_GUID_9473BECE_526D_34AA_1C97_88FE3EFAE71A'}
	(* Search for object contours in a binary image and determine their hierarchical relationship. (expert function) *)
	FUNCTION F_VN_FindContourHierarchyExp : HRESULT
	VAR_INPUT
		ipSrcImage	:	ITcVnImage;	(* Source image (1 channel, binary) *)
		ipContours	:	REFERENCE TO ITcVnContainer;	(* Returns a container which is filled with the found contours (ContainerType_Vector_Vector_TcVnPoint2_DINT; The elements of this container are single contours. Non-zero interface pointers are reused.) *)
		ipHierarchy	:	REFERENCE TO ITcVnContainer;	(* Returns a container which is filled with information on the found contours' hierarchy (ContainerType_Vector_TcVnVector4_DINT; The elements of this container are four-dimensional vectors containing the 0-based indices of the next [0] and the previous contour [1] at the same level, the first child [2], and the parent [3]. Non-zero interface pointers are reused.) *)
		eRetrievalMode	:	ETcVnContourRetrievalMode;	(* Specifies which contours are retrieved and how their relationship is encoded *)
		eApproximationMethod	:	ETcVnContourApproximationMethod;	(* Contour encoding *)
		aOffset	:	REFERENCE TO TcVnPoint;	(* Offset by which every contour point is shifted *)
		hrPrev	:	HRESULT;	(* HRESULT indicating the result of previous operations (If SUCCEEDED(hrPrev) equals false, no operation is executed.) *)
	END_VAR

END_FUNCTION

// Functions/Image Analysis/Object Detection/F_VN_FindContours

	{attribute 'TcIecLibraryType'}
	{attribute 'external_name' := 'F_VN_FindContours_GUID_FCB893B9_E591_3799_2A0C_20BA26051DE9'}
	(* Search for object contours in a binary image. Returns only external contours. *)
	FUNCTION F_VN_FindContours : HRESULT
	VAR_INPUT
		ipSrcImage	:	ITcVnImage;	(* Source image (1 channel, binary) *)
		ipContours	:	REFERENCE TO ITcVnContainer;	(* Returns a container which is filled with the found contours (ContainerType_Vector_Vector_TcVnPoint2_DINT; The elements of this container are single contours. Non-zero interface pointers are reused.) *)
		hrPrev	:	HRESULT;	(* HRESULT indicating the result of previous operations (If SUCCEEDED(hrPrev) equals false, no operation is executed.) *)
	END_VAR

END_FUNCTION

// Functions/Image Analysis/Object Detection/F_VN_FindContoursExp

	{attribute 'TcIecLibraryType'}
	{attribute 'external_name' := 'F_VN_FindContoursExp_GUID_8CBA5025_8ECB_358F_0E17_DE22AB7A2587'}
	(* Search for object contours in a binary image. (expert function) *)
	FUNCTION F_VN_FindContoursExp : HRESULT
	VAR_INPUT
		ipSrcImage	:	ITcVnImage;	(* Source image (1 channel, binary) *)
		ipContours	:	REFERENCE TO ITcVnContainer;	(* Returns a container which is filled with the found contours (ContainerType_Vector_Vector_TcVnPoint2_DINT; The elements of this container are single contours. Non-zero interface pointers are reused.) *)
		eRetrievalMode	:	ETcVnContourRetrievalMode;	(* Specifies which contours are retrieved and how their relationship is encoded *)
		eApproximationMethod	:	ETcVnContourApproximationMethod;	(* Contour encoding *)
		aOffset	:	REFERENCE TO TcVnPoint;	(* Offset by which every contour point is shifted *)
		hrPrev	:	HRESULT;	(* HRESULT indicating the result of previous operations (If SUCCEEDED(hrPrev) equals false, no operation is executed.) *)
	END_VAR

END_FUNCTION

// Functions/Image Analysis/Object Detection/F_VN_HoughCircles

	{attribute 'TcIecLibraryType'}
	{attribute 'external_name' := 'F_VN_HoughCircles_GUID_C629D5C8_F15A_3685_3EE3_DABA5DA8EF57'}
	(* Search for circles using the Hough transform. *)
	FUNCTION F_VN_HoughCircles : HRESULT
	VAR_INPUT
		ipSrcImage	:	ITcVnImage;	(* Source image (USINT, 1 channel, gray-level) *)
		ipCircles	:	REFERENCE TO ITcVnContainer;	(* Returns a container which is filled with the found circles (ContainerType_Vector_TcVnVector3_REAL; Each container element contains the x coordinate of the circle center [0], the y coordinate of the circle center [1], and the radius [2], respectively. Non-zero interface pointers are reused.) *)
		fInvAccuRatio	:	LREAL;	(* Inverted ratio of the accumulator size in relation to the source image's size (must be > 0. A value of 2 means that the size is halved in both directions.) *)
		fMinDist	:	LREAL;	(* Smallest allowed distance of two circles (must be > 0) *)
		hrPrev	:	HRESULT;	(* HRESULT indicating the result of previous operations (If SUCCEEDED(hrPrev) equals false, no operation is executed.) *)
	END_VAR

END_FUNCTION

// Functions/Image Analysis/Object Detection/F_VN_HoughCirclesExp

	{attribute 'TcIecLibraryType'}
	{attribute 'external_name' := 'F_VN_HoughCirclesExp_GUID_F105B70A_1E4C_3D67_2153_0BAD535BB162'}
	(* Search for circles using the Hough transform. (expert function) *)
	FUNCTION F_VN_HoughCirclesExp : HRESULT
	VAR_INPUT
		ipSrcImage	:	ITcVnImage;	(* Source image (USINT, 1 channel, gray-level) *)
		ipCircles	:	REFERENCE TO ITcVnContainer;	(* Returns a container which is filled with the found circles (ContainerType_Vector_TcVnVector3_REAL; Each container element contains the x coordinate of the circle center [0], the y coordinate of the circle center [1], and the radius [2], respectively. Non-zero interface pointers are reused.) *)
		fInvAccuRatio	:	LREAL;	(* Inverted ratio of the accumulator size in relation to the source image's size (must be > 0. A value of 2 means that the size is halved in both directions.) *)
		fMinDist	:	LREAL;	(* Smallest allowed distance of two circles (must be > 0) *)
		eHoughMethod	:	ETcVnHoughMethod;	(* Hough method to use (GRADIENT or GRADIENT_ALT) *)
		fParam1	:	LREAL;	(* First method specific parameter (GRADIENT, GRADIENT_ALT: upper threshold for canny edge detection, which must be > 0) *)
		fParam2	:	LREAL;	(* Second method specific parameter (GRADIENT: accumulator threshold for detecting circle centers, which must be > 0. GRADIENT_ALT: required circle perfectness, which must be > 0 and < 1, 1 would be a perfect circle) *)
		nMinRadius	:	UDINT;	(* Minimum circle radius allowed *)
		nMaxRadius	:	UDINT;	(* Maximum circle radius allowed (if 0, the value is internally set to max(image rows, image columns)) *)
		hrPrev	:	HRESULT;	(* HRESULT indicating the result of previous operations (If SUCCEEDED(hrPrev) equals false, no operation is executed.) *)
	END_VAR

END_FUNCTION

// Functions/Image Analysis/Object Detection/F_VN_HoughLines

	{attribute 'TcIecLibraryType'}
	{attribute 'external_name' := 'F_VN_HoughLines_GUID_769839FF_1529_3A59_2422_8F8DC7D5C4E7'}
	(* Search for lines using the standard Hough transform. *)
	FUNCTION F_VN_HoughLines : HRESULT
	VAR_INPUT
		ipSrcImage	:	ITcVnImage;	(* Source image (USINT, 1 channel, binary, may be modified by the function) *)
		ipLines	:	REFERENCE TO ITcVnContainer;	(* Returns a container which is filled with the found lines (ContainerType_Vector_TcVnVector2_REAL; Each container element contains the distance from the origin [0] in pixels and the rotation angle [1] in radians, respectively. Non-zero interface pointers are reused.) *)
		fDistRes	:	LREAL;	(* Distance resolution of the accumulator (in pixels, must be > 0) *)
		fAngleRes	:	LREAL;	(* Angle resolution of the accumulator (in radians, must be > 0) *)
		nAccuThreshold	:	UDINT;	(* Accumulator threshold *)
		hrPrev	:	HRESULT;	(* HRESULT indicating the result of previous operations (If SUCCEEDED(hrPrev) equals false, no operation is executed.) *)
	END_VAR

END_FUNCTION

// Functions/Image Analysis/Object Detection/F_VN_HoughLinesExp

	{attribute 'TcIecLibraryType'}
	{attribute 'external_name' := 'F_VN_HoughLinesExp_GUID_5C4615B1_87D1_3BCB_3949_4D4FB5C5EED7'}
	(* Search for lines using the standard Hough transform. (expert function) *)
	FUNCTION F_VN_HoughLinesExp : HRESULT
	VAR_INPUT
		ipSrcImage	:	ITcVnImage;	(* Source image (USINT, 1 channel, binary, may be modified by the function) *)
		ipLines	:	REFERENCE TO ITcVnContainer;	(* Returns a container which is filled with the found lines (ContainerType_Vector_TcVnVector2_REAL; Each container element contains the distance from the origin [0] in pixels and the rotation angle [1] in radians, respectively. Non-zero interface pointers are reused.) *)
		fDistRes	:	LREAL;	(* Distance resolution of the accumulator (in pixels, must be > 0) *)
		fAngleRes	:	LREAL;	(* Angle resolution of the accumulator (in radians, must be > 0) *)
		nAccuThreshold	:	UDINT;	(* Accumulator threshold *)
		fDistResDiv	:	LREAL;	(* Divisor of the distance resolution for the multi-scale Hough transform (>= 0, must be > 0 if fAngleResDiv is > 0) *)
		fAngleResDiv	:	LREAL;	(* Divisor of the angle resolution for the multi-scale Hough transform (>= 0, must be > 0 if fDistResDiv is > 0) *)
		hrPrev	:	HRESULT;	(* HRESULT indicating the result of previous operations (If SUCCEEDED(hrPrev) equals false, no operation is executed.) *)
	END_VAR

END_FUNCTION

// Functions/Image Analysis/Object Detection/F_VN_HoughLinesP

	{attribute 'TcIecLibraryType'}
	{attribute 'external_name' := 'F_VN_HoughLinesP_GUID_A285A5D8_D627_316D_1A81_C3435631D87E'}
	(* Search for line segments using the probabilistic Hough transform. *)
	FUNCTION F_VN_HoughLinesP : HRESULT
	VAR_INPUT
		ipSrcImage	:	ITcVnImage;	(* Source image (USINT, 1 channel, binary, may be modified by the function) *)
		ipLines	:	REFERENCE TO ITcVnContainer;	(* Returns a container which is filled with the found line segments (ContainerType_Vector_TcVnVector4_DINT; Each container element contains the two ending points. Non-zero interface pointers are reused.) *)
		fDistRes	:	LREAL;	(* Distance resolution of the accumulator (in pixels, must be > 0) *)
		fAngleRes	:	LREAL;	(* Angle resolution of the accumulator (in radians, must be > 0) *)
		nAccuThreshold	:	UDINT;	(* Accumulator threshold *)
		hrPrev	:	HRESULT;	(* HRESULT indicating the result of previous operations (If SUCCEEDED(hrPrev) equals false, no operation is executed.) *)
	END_VAR

END_FUNCTION

// Functions/Image Analysis/Object Detection/F_VN_HoughLinesPExp

	{attribute 'TcIecLibraryType'}
	{attribute 'external_name' := 'F_VN_HoughLinesPExp_GUID_2FECC39D_3C18_3020_3E7D_3EEC049DFC4C'}
	(* Search for line segments using the probabilistic Hough transform. (expert function) *)
	FUNCTION F_VN_HoughLinesPExp : HRESULT
	VAR_INPUT
		ipSrcImage	:	ITcVnImage;	(* Source image (USINT, 1 channel, binary, may be modified by the function) *)
		ipLines	:	REFERENCE TO ITcVnContainer;	(* Returns a container which is filled with the found line segments (ContainerType_Vector_TcVnVector4_DINT; Each container element contains the two ending points. Non-zero interface pointers are reused.) *)
		fDistRes	:	LREAL;	(* Distance resolution of the accumulator (in pixels, must be > 0) *)
		fAngleRes	:	LREAL;	(* Angle resolution of the accumulator (in radians, must be > 0) *)
		nAccuThreshold	:	UDINT;	(* Accumulator threshold *)
		fMinLineLength	:	LREAL;	(* Minimum line length to search for *)
		fMaxLineGap	:	LREAL;	(* Maximum gap between points on the same line *)
		hrPrev	:	HRESULT;	(* HRESULT indicating the result of previous operations (If SUCCEEDED(hrPrev) equals false, no operation is executed.) *)
	END_VAR

END_FUNCTION

// Functions/Image Analysis/Object Detection/F_VN_MatchImageHuMoments

	{attribute 'TcIecLibraryType'}
	{attribute 'external_name' := 'F_VN_MatchImageHuMoments_GUID_91AD0F22_BBF2_318D_374F_D21932268E6B'}
	(* Compare two images using the Hu moment invariants. *)
	FUNCTION F_VN_MatchImageHuMoments : HRESULT
	VAR_INPUT
		ipImage1	:	ITcVnImage;	(* First image (1 channel) *)
		ipImage2	:	ITcVnImage;	(* Second image (1 channel) *)
		eComparisonMethod	:	ETcVnContoursMatchComparisonMethod;	(* Method used for comparing the Hu moment invariants of the images *)
		fDissimilarity	:	REFERENCE TO LREAL;	(* Returns the dissimilarity of the image Hu moment invariants depending on the chosen comparison method *)
		hrPrev	:	HRESULT;	(* HRESULT indicating the result of previous operations (If SUCCEEDED(hrPrev) equals false, no operation is executed.) *)
	END_VAR

END_FUNCTION

// Functions/Image Analysis/Object Detection/F_VN_MatchTemplate

	{attribute 'TcIecLibraryType'}
	{attribute 'external_name' := 'F_VN_MatchTemplate_GUID_34C2D7EC_1AA6_34B0_369D_70306E781324'}
	(* Match a template image with every location in the source image (using the TCVN_TMM_CCORR_NORMED method) and save the comparison results. *)
	FUNCTION F_VN_MatchTemplate : HRESULT
	VAR_INPUT
		ipSrcImage	:	ITcVnImage;	(* Source image (USINT or REAL, 1 or 3 channels) *)
		ipTemplateImage	:	ITcVnImage;	(* Template image (same type as ipSrcImage, smaller width and height) *)
		ipResultImage	:	REFERENCE TO ITcVnImage;	(* Returns the result image (REAL, normalized to [0..1], 1 channel, dimensions: (ipSrcImage.width - ipTemplateImage.width + 1) x (ipSrcImage.height - ipTemplateImage.height + 1). The best match is the global maximum. The position in ipResultImage is the top-left corner of ipTemplateImage position in ipSrcImage) *)
		hrPrev	:	HRESULT;	(* HRESULT indicating the result of previous operations (If SUCCEEDED(hrPrev) equals false, no operation is executed.) *)
	END_VAR

END_FUNCTION

// Functions/Image Analysis/Object Detection/F_VN_MatchTemplateExp

	{attribute 'TcIecLibraryType'}
	{attribute 'external_name' := 'F_VN_MatchTemplateExp_GUID_C2A9E07A_3473_360D_0D6A_F1D92C10869B'}
	(* Match a template image with every location in the source image and save the comparison results. (expert function) *)
	FUNCTION F_VN_MatchTemplateExp : HRESULT
	VAR_INPUT
		ipSrcImage	:	ITcVnImage;	(* Source image (USINT or REAL, 1 or 3 channels) *)
		ipTemplateImage	:	ITcVnImage;	(* Template image (same type as ipSrcImage, smaller width and height) *)
		ipResultImage	:	REFERENCE TO ITcVnImage;	(* Returns the result image (REAL, 1 channel, dimensions: (ipSrcImage.width - ipTemplateImage.width + 1) x (ipSrcImage.height - ipTemplateImage.height + 1). The best match is the global minimum (SQDIFF(_NORMED)) or maximum (CCORR(_NORMED), CCOEFF(_NORMED)). The position in ipResultImage is the top-left corner of ipTemplateImage position in ipSrcImage) *)
		eMatchMethod	:	ETcVnTemplateMatchMethod;	(* Specifies the template match method *)
		ipTemplateMask	:	ITcVnImage;	(* Optional mask for ipTemplateImage (only supported for SQDIFF and CCORR_NORMED, same type and size as ipTemplateImage) *)
		hrPrev	:	HRESULT;	(* HRESULT indicating the result of previous operations (If SUCCEEDED(hrPrev) equals false, no operation is executed.) *)
	END_VAR

END_FUNCTION

// Functions/Image Analysis/Object Detection/F_VN_MatchTemplateAndEvaluate

	{attribute 'TcIecLibraryType'}
	{attribute 'external_name' := 'F_VN_MatchTemplateAndEvaluate_GUID_20BF5AED_16A1_36AF_37C8_F4BC340C96B4'}
	(* Match a template image with every location in the source image (using the TCVN_TMM_CCORR_NORMED method) and evaluate the comparison results. Returns a sorted list of possible matches (best match first). *)
	FUNCTION F_VN_MatchTemplateAndEvaluate : HRESULT
	VAR_INPUT
		ipSrcImage	:	ITcVnImage;	(* Source image (USINT or REAL, 1 or 3 channels) *)
		ipTemplateImage	:	ITcVnImage;	(* Template image (same type as ipSrcImage, smaller width and height) *)
		ipMatches	:	REFERENCE TO ITcVnContainer;	(* Returns the matching positions (ContainerType_Vector_TcVnPoint2_DINT, where each element represents the top-left corner of ipTemplateImage) in ipSrcImage, sorted by relevance (best match first) *)
		fMatchThreshold	:	REAL;	(* Threshold to separate relevant from irrelevant matches (0..1, 1.0  would be a perfect match. To find a suitable value, you could evaluate some sample result images of F_VN_MatchTemplate.) *)
		hrPrev	:	HRESULT;	(* HRESULT indicating the result of previous operations (If SUCCEEDED(hrPrev) equals false, no operation is executed.) *)
	END_VAR

END_FUNCTION

// Functions/Image Analysis/Object Detection/F_VN_MatchTemplateAndEvaluateExp

	{attribute 'TcIecLibraryType'}
	{attribute 'external_name' := 'F_VN_MatchTemplateAndEvaluateExp_GUID_A65635BE_BD93_34F5_0F03_6F7EA4633A05'}
	(* Match a template image with every location in the source image and evaluate the comparison results. Returns a sorted list of possible matches (best match first). (expert function) *)
	FUNCTION F_VN_MatchTemplateAndEvaluateExp : HRESULT
	VAR_INPUT
		ipSrcImage	:	ITcVnImage;	(* Source image (USINT or REAL, 1 or 3 channels) *)
		ipTemplateImage	:	ITcVnImage;	(* Template image (same type as ipSrcImage, smaller width and height) *)
		ipMatches	:	REFERENCE TO ITcVnContainer;	(* Returns the matching positions (ContainerType_Vector_TcVnPoint2_DINT, where each element represents the top-left corner of ipTemplateImage) in ipSrcImage, sorted by relevance (best match first) *)
		fMatchThreshold	:	REAL;	(* Threshold to separate relevant from irrelevant matches (0..1 for NORMED methods, otherwise dependent on template size and content. To find a suitable value, you could evaluate some sample result images of F_VN_MatchTemplateExp.) *)
		eMatchMethod	:	ETcVnTemplateMatchMethod;	(* Specifies the template match method *)
		ipTemplateMask	:	ITcVnImage;	(* Optional mask for ipTemplateImage (only supported for SQDIFF and CCORR_NORMED, same type and size as ipTemplateImage) *)
		fScaleFactor	:	REAL;	(* Factor (0..1] to reduce source and template image width and height for better performance (but less accuracy!) *)
		eInterpolationType	:	ETcVnInterpolationType;	(* Image resize interpolation type (only used if fScaleFactor != 1, TCVN_IT_BILINEAR recommended for most cases) *)
		ipMatchValues	:	REFERENCE TO ITcVnContainer;	(* Optionally returns the matching values (ContainerType_Vector_REAL, same size and sort order as ipMatches. Set to 0 if not required.) *)
		hrPrev	:	HRESULT;	(* HRESULT indicating the result of previous operations (If SUCCEEDED(hrPrev) equals false, no operation is executed.) *)
	END_VAR

END_FUNCTION

// Functions/Basic Container Operations/F_VN_AppendToContainer/F_VN_AppendToContainer_ITcVnContainer

	{attribute 'TcIecLibraryType'}
	{attribute 'external_name' := 'F_VN_AppendToContainer_ITcVnContainer_GUID_FC50B7C8_99F9_30A5_262C_2E86E2E59366'}
	(* Append a single element to a container or concatenate containers (if ipElement has the same typeId as ipContainer). *)
	FUNCTION F_VN_AppendToContainer_ITcVnContainer : HRESULT
	VAR_INPUT
		ipElement	:	ITcVnContainer;	(* Single element to append to ipContainer or container with several elements to be concatenated *)
		ipContainer	:	ITcVnContainer;	(* Container to which the element(s) will be appended *)
		hrPrev	:	HRESULT;	(* HRESULT indicating the result of previous operations (If SUCCEEDED(hrPrev) equals false, no operation is executed.) *)
	END_VAR

END_FUNCTION

// Functions/Basic Container Operations/F_VN_AppendToContainer/F_VN_AppendToContainer_ITcVnForwardIterator

	{attribute 'TcIecLibraryType'}
	{attribute 'external_name' := 'F_VN_AppendToContainer_ITcVnForwardIterator_GUID_9CDF5DEA_059D_3205_0E72_5BDBE2F64E63'}
	(* Append a single element (represented by an iterator)to a container. *)
	FUNCTION F_VN_AppendToContainer_ITcVnForwardIterator : HRESULT
	VAR_INPUT
		ipElement	:	ITcVnForwardIterator;	(* Single element to append to ipContainer *)
		ipContainer	:	ITcVnContainer;	(* Container to which the element(s) will be appended *)
		hrPrev	:	HRESULT;	(* HRESULT indicating the result of previous operations (If SUCCEEDED(hrPrev) equals false, no operation is executed.) *)
	END_VAR

END_FUNCTION

// Functions/Basic Container Operations/F_VN_AppendToContainer/F_VN_AppendToContainer_DINT

	{attribute 'TcIecLibraryType'}
	{attribute 'external_name' := 'F_VN_AppendToContainer_DINT_GUID_31C28DF3_E36B_3208_17A0_A6C1B2E60765'}
	(* Append a single element of type DINT to a container. *)
	FUNCTION F_VN_AppendToContainer_DINT : HRESULT
	VAR_INPUT
		nElement	:	DINT;	(* Single element to append to ipContainer *)
		ipContainer	:	ITcVnContainer;	(* Container to which the element will be appended *)
		hrPrev	:	HRESULT;	(* HRESULT indicating the result of previous operations (If SUCCEEDED(hrPrev) equals false, no operation is executed.) *)
	END_VAR

END_FUNCTION

// Functions/Basic Container Operations/F_VN_AppendToContainer/F_VN_AppendToContainer_INT

	{attribute 'TcIecLibraryType'}
	{attribute 'external_name' := 'F_VN_AppendToContainer_INT_GUID_EB831201_87E6_336A_0A16_8AE03B275570'}
	(* Append a single element of type INT to a container. *)
	FUNCTION F_VN_AppendToContainer_INT : HRESULT
	VAR_INPUT
		nElement	:	INT;	(* Single element to append to ipContainer *)
		ipContainer	:	ITcVnContainer;	(* Container to which the element will be appended *)
		hrPrev	:	HRESULT;	(* HRESULT indicating the result of previous operations (If SUCCEEDED(hrPrev) equals false, no operation is executed.) *)
	END_VAR

END_FUNCTION

// Functions/Basic Container Operations/F_VN_AppendToContainer/F_VN_AppendToContainer_LREAL

	{attribute 'TcIecLibraryType'}
	{attribute 'external_name' := 'F_VN_AppendToContainer_LREAL_GUID_C60F93DB_4076_3ED0_2221_23F8A2771A5F'}
	(* Append a single element of type LREAL to a container. *)
	FUNCTION F_VN_AppendToContainer_LREAL : HRESULT
	VAR_INPUT
		fElement	:	LREAL;	(* Single element to append to ipContainer *)
		ipContainer	:	ITcVnContainer;	(* Container to which the element will be appended *)
		hrPrev	:	HRESULT;	(* HRESULT indicating the result of previous operations (If SUCCEEDED(hrPrev) equals false, no operation is executed.) *)
	END_VAR

END_FUNCTION

// Functions/Basic Container Operations/F_VN_AppendToContainer/F_VN_AppendToContainer_REAL

	{attribute 'TcIecLibraryType'}
	{attribute 'external_name' := 'F_VN_AppendToContainer_REAL_GUID_DF0A4B84_0BB1_3824_3BA5_E668C13985F5'}
	(* Append a single element of type REAL to a container. *)
	FUNCTION F_VN_AppendToContainer_REAL : HRESULT
	VAR_INPUT
		fElement	:	REAL;	(* Single element to append to ipContainer *)
		ipContainer	:	ITcVnContainer;	(* Container to which the element will be appended *)
		hrPrev	:	HRESULT;	(* HRESULT indicating the result of previous operations (If SUCCEEDED(hrPrev) equals false, no operation is executed.) *)
	END_VAR

END_FUNCTION

// Functions/Basic Container Operations/F_VN_AppendToContainer/F_VN_AppendToContainer_SINT

	{attribute 'TcIecLibraryType'}
	{attribute 'external_name' := 'F_VN_AppendToContainer_SINT_GUID_592FDA8E_B93A_348E_3F42_8BB17F823087'}
	(* Append a single element of type SINT to a container. *)
	FUNCTION F_VN_AppendToContainer_SINT : HRESULT
	VAR_INPUT
		nElement	:	SINT;	(* Single element to append to ipContainer *)
		ipContainer	:	ITcVnContainer;	(* Container to which the element will be appended *)
		hrPrev	:	HRESULT;	(* HRESULT indicating the result of previous operations (If SUCCEEDED(hrPrev) equals false, no operation is executed.) *)
	END_VAR

END_FUNCTION

// Functions/Basic Container Operations/F_VN_AppendToContainer/F_VN_AppendToContainer_TcVnDMatch

	{attribute 'TcIecLibraryType'}
	{attribute 'external_name' := 'F_VN_AppendToContainer_TcVnDMatch_GUID_4329EEF1_FD6D_3301_3211_09D923A76879'}
	(* Append a single element of type TcVnDMatch to a container. *)
	FUNCTION F_VN_AppendToContainer_TcVnDMatch : HRESULT
	VAR_INPUT
		stElement	:	REFERENCE TO TcVnDMatch;	(* Single element to append to ipContainer *)
		ipContainer	:	ITcVnContainer;	(* Container to which the element will be appended *)
		hrPrev	:	HRESULT;	(* HRESULT indicating the result of previous operations (If SUCCEEDED(hrPrev) equals false, no operation is executed.) *)
	END_VAR

END_FUNCTION

// Functions/Basic Container Operations/F_VN_AppendToContainer/F_VN_AppendToContainer_TcVnKeyPoint

	{attribute 'TcIecLibraryType'}
	{attribute 'external_name' := 'F_VN_AppendToContainer_TcVnKeyPoint_GUID_AAB1ED15_D350_3622_2782_B39F421ADC95'}
	(* Append a single element of type TcVnKeyPoint to a container. *)
	FUNCTION F_VN_AppendToContainer_TcVnKeyPoint : HRESULT
	VAR_INPUT
		stElement	:	REFERENCE TO TcVnKeyPoint;	(* Single element to append to ipContainer *)
		ipContainer	:	ITcVnContainer;	(* Container to which the element will be appended *)
		hrPrev	:	HRESULT;	(* HRESULT indicating the result of previous operations (If SUCCEEDED(hrPrev) equals false, no operation is executed.) *)
	END_VAR

END_FUNCTION

// Functions/Basic Container Operations/F_VN_AppendToContainer/F_VN_AppendToContainer_TcVnPoint2_DINT

	{attribute 'TcIecLibraryType'}
	{attribute 'external_name' := 'F_VN_AppendToContainer_TcVnPoint2_DINT_GUID_959B578D_4793_3FB4_154D_46966D3C179F'}
	(* Append a single element of type TcVnPoint2_DINT to a container. *)
	FUNCTION F_VN_AppendToContainer_TcVnPoint2_DINT : HRESULT
	VAR_INPUT
		aElement	:	REFERENCE TO TcVnPoint2_DINT;	(* Single element to append to ipContainer *)
		ipContainer	:	ITcVnContainer;	(* Container to which the element will be appended *)
		hrPrev	:	HRESULT;	(* HRESULT indicating the result of previous operations (If SUCCEEDED(hrPrev) equals false, no operation is executed.) *)
	END_VAR

END_FUNCTION

// Functions/Basic Container Operations/F_VN_AppendToContainer/F_VN_AppendToContainer_TcVnPoint2_LREAL

	{attribute 'TcIecLibraryType'}
	{attribute 'external_name' := 'F_VN_AppendToContainer_TcVnPoint2_LREAL_GUID_6159B5AB_3C3D_3662_0DD6_902D18483C54'}
	(* Append a single element of type TcVnPoint2_LREAL to a container. *)
	FUNCTION F_VN_AppendToContainer_TcVnPoint2_LREAL : HRESULT
	VAR_INPUT
		aElement	:	REFERENCE TO TcVnPoint2_LREAL;	(* Single element to append to ipContainer *)
		ipContainer	:	ITcVnContainer;	(* Container to which the element will be appended *)
		hrPrev	:	HRESULT;	(* HRESULT indicating the result of previous operations (If SUCCEEDED(hrPrev) equals false, no operation is executed.) *)
	END_VAR

END_FUNCTION

// Functions/Basic Container Operations/F_VN_AppendToContainer/F_VN_AppendToContainer_TcVnPoint2_REAL

	{attribute 'TcIecLibraryType'}
	{attribute 'external_name' := 'F_VN_AppendToContainer_TcVnPoint2_REAL_GUID_D88DD509_40A4_322C_26A0_36F9347B3C1E'}
	(* Append a single element of type TcVnPoint2_REAL to a container. *)
	FUNCTION F_VN_AppendToContainer_TcVnPoint2_REAL : HRESULT
	VAR_INPUT
		aElement	:	REFERENCE TO TcVnPoint2_REAL;	(* Single element to append to ipContainer *)
		ipContainer	:	ITcVnContainer;	(* Container to which the element will be appended *)
		hrPrev	:	HRESULT;	(* HRESULT indicating the result of previous operations (If SUCCEEDED(hrPrev) equals false, no operation is executed.) *)
	END_VAR

END_FUNCTION

// Functions/Basic Container Operations/F_VN_AppendToContainer/F_VN_AppendToContainer_TcVnPoint3_LREAL

	{attribute 'TcIecLibraryType'}
	{attribute 'external_name' := 'F_VN_AppendToContainer_TcVnPoint3_LREAL_GUID_342CD413_B0C5_3113_0758_3F5B37489530'}
	(* Append a single element of type TcVnPoint3_LREAL to a container. *)
	FUNCTION F_VN_AppendToContainer_TcVnPoint3_LREAL : HRESULT
	VAR_INPUT
		aElement	:	REFERENCE TO TcVnPoint3_LREAL;	(* Single element to append to ipContainer *)
		ipContainer	:	ITcVnContainer;	(* Container to which the element will be appended *)
		hrPrev	:	HRESULT;	(* HRESULT indicating the result of previous operations (If SUCCEEDED(hrPrev) equals false, no operation is executed.) *)
	END_VAR

END_FUNCTION

// Functions/Basic Container Operations/F_VN_AppendToContainer/F_VN_AppendToContainer_TcVnPoint3_REAL

	{attribute 'TcIecLibraryType'}
	{attribute 'external_name' := 'F_VN_AppendToContainer_TcVnPoint3_REAL_GUID_28F44627_F0F4_36AD_1B88_781A4C151607'}
	(* Append a single element of type TcVnPoint3_REAL to a container. *)
	FUNCTION F_VN_AppendToContainer_TcVnPoint3_REAL : HRESULT
	VAR_INPUT
		aElement	:	REFERENCE TO TcVnPoint3_REAL;	(* Single element to append to ipContainer *)
		ipContainer	:	ITcVnContainer;	(* Container to which the element will be appended *)
		hrPrev	:	HRESULT;	(* HRESULT indicating the result of previous operations (If SUCCEEDED(hrPrev) equals false, no operation is executed.) *)
	END_VAR

END_FUNCTION

// Functions/Basic Container Operations/F_VN_AppendToContainer/F_VN_AppendToContainer_TcVnRectangle_DINT

	{attribute 'TcIecLibraryType'}
	{attribute 'external_name' := 'F_VN_AppendToContainer_TcVnRectangle_DINT_GUID_308961C9_DF32_34EF_0D08_650464EE6AA4'}
	(* Append a single element of type TcVnRectangle_DINT to a container. *)
	FUNCTION F_VN_AppendToContainer_TcVnRectangle_DINT : HRESULT
	VAR_INPUT
		stElement	:	REFERENCE TO TcVnRectangle_DINT;	(* Single element to append to ipContainer *)
		ipContainer	:	ITcVnContainer;	(* Container to which the element will be appended *)
		hrPrev	:	HRESULT;	(* HRESULT indicating the result of previous operations (If SUCCEEDED(hrPrev) equals false, no operation is executed.) *)
	END_VAR

END_FUNCTION

// Functions/Basic Container Operations/F_VN_AppendToContainer/F_VN_AppendToContainer_TcVnVector2_DINT

	{attribute 'TcIecLibraryType'}
	{attribute 'external_name' := 'F_VN_AppendToContainer_TcVnVector2_DINT_GUID_B5923707_5908_356D_38CB_E49C103D9C8F'}
	(* Append a single element of type TcVnVector2_DINT to a container. *)
	FUNCTION F_VN_AppendToContainer_TcVnVector2_DINT : HRESULT
	VAR_INPUT
		aElement	:	REFERENCE TO TcVnVector2_DINT;	(* Single element to append to ipContainer *)
		ipContainer	:	ITcVnContainer;	(* Container to which the element will be appended *)
		hrPrev	:	HRESULT;	(* HRESULT indicating the result of previous operations (If SUCCEEDED(hrPrev) equals false, no operation is executed.) *)
	END_VAR

END_FUNCTION

// Functions/Basic Container Operations/F_VN_AppendToContainer/F_VN_AppendToContainer_TcVnVector2_INT

	{attribute 'TcIecLibraryType'}
	{attribute 'external_name' := 'F_VN_AppendToContainer_TcVnVector2_INT_GUID_F7387903_E97A_3B99_2033_4EB10D12A1E9'}
	(* Append a single element of type TcVnVector2_INT to a container. *)
	FUNCTION F_VN_AppendToContainer_TcVnVector2_INT : HRESULT
	VAR_INPUT
		aElement	:	REFERENCE TO TcVnVector2_INT;	(* Single element to append to ipContainer *)
		ipContainer	:	ITcVnContainer;	(* Container to which the element will be appended *)
		hrPrev	:	HRESULT;	(* HRESULT indicating the result of previous operations (If SUCCEEDED(hrPrev) equals false, no operation is executed.) *)
	END_VAR

END_FUNCTION

// Functions/Basic Container Operations/F_VN_AppendToContainer/F_VN_AppendToContainer_TcVnVector2_REAL

	{attribute 'TcIecLibraryType'}
	{attribute 'external_name' := 'F_VN_AppendToContainer_TcVnVector2_REAL_GUID_3E886E59_2AAE_34FF_26C8_FAD9FC2F5F83'}
	(* Append a single element of type TcVnVector2_REAL to a container. *)
	FUNCTION F_VN_AppendToContainer_TcVnVector2_REAL : HRESULT
	VAR_INPUT
		aElement	:	REFERENCE TO TcVnVector2_REAL;	(* Single element to append to ipContainer *)
		ipContainer	:	ITcVnContainer;	(* Container to which the element will be appended *)
		hrPrev	:	HRESULT;	(* HRESULT indicating the result of previous operations (If SUCCEEDED(hrPrev) equals false, no operation is executed.) *)
	END_VAR

END_FUNCTION

// Functions/Basic Container Operations/F_VN_AppendToContainer/F_VN_AppendToContainer_TcVnVector2_SINT

	{attribute 'TcIecLibraryType'}
	{attribute 'external_name' := 'F_VN_AppendToContainer_TcVnVector2_SINT_GUID_46623109_6DEE_3F6A_07A1_A4A3D7D28C0E'}
	(* Append a single element of type TcVnVector2_SINT to a container. *)
	FUNCTION F_VN_AppendToContainer_TcVnVector2_SINT : HRESULT
	VAR_INPUT
		aElement	:	REFERENCE TO TcVnVector2_SINT;	(* Single element to append to ipContainer *)
		ipContainer	:	ITcVnContainer;	(* Container to which the element will be appended *)
		hrPrev	:	HRESULT;	(* HRESULT indicating the result of previous operations (If SUCCEEDED(hrPrev) equals false, no operation is executed.) *)
	END_VAR

END_FUNCTION

// Functions/Basic Container Operations/F_VN_AppendToContainer/F_VN_AppendToContainer_TcVnVector2_UINT

	{attribute 'TcIecLibraryType'}
	{attribute 'external_name' := 'F_VN_AppendToContainer_TcVnVector2_UINT_GUID_91EBFA64_CBE2_3CA7_3555_07DD4A650409'}
	(* Append a single element of type TcVnVector2_UINT to a container. *)
	FUNCTION F_VN_AppendToContainer_TcVnVector2_UINT : HRESULT
	VAR_INPUT
		aElement	:	REFERENCE TO TcVnVector2_UINT;	(* Single element to append to ipContainer *)
		ipContainer	:	ITcVnContainer;	(* Container to which the element will be appended *)
		hrPrev	:	HRESULT;	(* HRESULT indicating the result of previous operations (If SUCCEEDED(hrPrev) equals false, no operation is executed.) *)
	END_VAR

END_FUNCTION

// Functions/Basic Container Operations/F_VN_AppendToContainer/F_VN_AppendToContainer_TcVnVector2_USINT

	{attribute 'TcIecLibraryType'}
	{attribute 'external_name' := 'F_VN_AppendToContainer_TcVnVector2_USINT_GUID_3BFF2E2F_550D_3AE9_3606_243D4CD1F210'}
	(* Append a single element of type TcVnVector2_USINT to a container. *)
	FUNCTION F_VN_AppendToContainer_TcVnVector2_USINT : HRESULT
	VAR_INPUT
		aElement	:	REFERENCE TO TcVnVector2_USINT;	(* Single element to append to ipContainer *)
		ipContainer	:	ITcVnContainer;	(* Container to which the element will be appended *)
		hrPrev	:	HRESULT;	(* HRESULT indicating the result of previous operations (If SUCCEEDED(hrPrev) equals false, no operation is executed.) *)
	END_VAR

END_FUNCTION

// Functions/Basic Container Operations/F_VN_AppendToContainer/F_VN_AppendToContainer_TcVnVector3_INT

	{attribute 'TcIecLibraryType'}
	{attribute 'external_name' := 'F_VN_AppendToContainer_TcVnVector3_INT_GUID_727F30D4_3D86_328A_330A_38884EAE3D59'}
	(* Append a single element of type TcVnVector3_INT to a container. *)
	FUNCTION F_VN_AppendToContainer_TcVnVector3_INT : HRESULT
	VAR_INPUT
		aElement	:	REFERENCE TO TcVnVector3_INT;	(* Single element to append to ipContainer *)
		ipContainer	:	ITcVnContainer;	(* Container to which the element will be appended *)
		hrPrev	:	HRESULT;	(* HRESULT indicating the result of previous operations (If SUCCEEDED(hrPrev) equals false, no operation is executed.) *)
	END_VAR

END_FUNCTION

// Functions/Basic Container Operations/F_VN_AppendToContainer/F_VN_AppendToContainer_TcVnVector3_REAL

	{attribute 'TcIecLibraryType'}
	{attribute 'external_name' := 'F_VN_AppendToContainer_TcVnVector3_REAL_GUID_26ED8719_A6F2_32D1_16B0_D8114649C505'}
	(* Append a single element of type TcVnVector3_REAL to a container. *)
	FUNCTION F_VN_AppendToContainer_TcVnVector3_REAL : HRESULT
	VAR_INPUT
		aElement	:	REFERENCE TO TcVnVector3_REAL;	(* Single element to append to ipContainer *)
		ipContainer	:	ITcVnContainer;	(* Container to which the element will be appended *)
		hrPrev	:	HRESULT;	(* HRESULT indicating the result of previous operations (If SUCCEEDED(hrPrev) equals false, no operation is executed.) *)
	END_VAR

END_FUNCTION

// Functions/Basic Container Operations/F_VN_AppendToContainer/F_VN_AppendToContainer_TcVnVector3_SINT

	{attribute 'TcIecLibraryType'}
	{attribute 'external_name' := 'F_VN_AppendToContainer_TcVnVector3_SINT_GUID_349569D3_D1E9_30E4_3FF0_83391A4BDBB4'}
	(* Append a single element of type TcVnVector3_SINT to a container. *)
	FUNCTION F_VN_AppendToContainer_TcVnVector3_SINT : HRESULT
	VAR_INPUT
		aElement	:	REFERENCE TO TcVnVector3_SINT;	(* Single element to append to ipContainer *)
		ipContainer	:	ITcVnContainer;	(* Container to which the element will be appended *)
		hrPrev	:	HRESULT;	(* HRESULT indicating the result of previous operations (If SUCCEEDED(hrPrev) equals false, no operation is executed.) *)
	END_VAR

END_FUNCTION

// Functions/Basic Container Operations/F_VN_AppendToContainer/F_VN_AppendToContainer_TcVnVector3_UINT

	{attribute 'TcIecLibraryType'}
	{attribute 'external_name' := 'F_VN_AppendToContainer_TcVnVector3_UINT_GUID_022337F8_1AD4_3D89_0A5A_C6911AE9819B'}
	(* Append a single element of type TcVnVector3_UINT to a container. *)
	FUNCTION F_VN_AppendToContainer_TcVnVector3_UINT : HRESULT
	VAR_INPUT
		aElement	:	REFERENCE TO TcVnVector3_UINT;	(* Single element to append to ipContainer *)
		ipContainer	:	ITcVnContainer;	(* Container to which the element will be appended *)
		hrPrev	:	HRESULT;	(* HRESULT indicating the result of previous operations (If SUCCEEDED(hrPrev) equals false, no operation is executed.) *)
	END_VAR

END_FUNCTION

// Functions/Basic Container Operations/F_VN_AppendToContainer/F_VN_AppendToContainer_TcVnVector3_USINT

	{attribute 'TcIecLibraryType'}
	{attribute 'external_name' := 'F_VN_AppendToContainer_TcVnVector3_USINT_GUID_7F438F28_F7C5_3254_260D_8557E123F477'}
	(* Append a single element of type TcVnVector3_USINT to a container. *)
	FUNCTION F_VN_AppendToContainer_TcVnVector3_USINT : HRESULT
	VAR_INPUT
		aElement	:	REFERENCE TO TcVnVector3_USINT;	(* Single element to append to ipContainer *)
		ipContainer	:	ITcVnContainer;	(* Container to which the element will be appended *)
		hrPrev	:	HRESULT;	(* HRESULT indicating the result of previous operations (If SUCCEEDED(hrPrev) equals false, no operation is executed.) *)
	END_VAR

END_FUNCTION

// Functions/Basic Container Operations/F_VN_AppendToContainer/F_VN_AppendToContainer_TcVnVector4_DINT

	{attribute 'TcIecLibraryType'}
	{attribute 'external_name' := 'F_VN_AppendToContainer_TcVnVector4_DINT_GUID_7F929A89_D061_3C67_3D60_5478F06D2AEA'}
	(* Append a single element of type TcVnVector4_DINT to a container. *)
	FUNCTION F_VN_AppendToContainer_TcVnVector4_DINT : HRESULT
	VAR_INPUT
		aElement	:	REFERENCE TO TcVnVector4_DINT;	(* Single element to append to ipContainer *)
		ipContainer	:	ITcVnContainer;	(* Container to which the element will be appended *)
		hrPrev	:	HRESULT;	(* HRESULT indicating the result of previous operations (If SUCCEEDED(hrPrev) equals false, no operation is executed.) *)
	END_VAR

END_FUNCTION

// Functions/Basic Container Operations/F_VN_AppendToContainer/F_VN_AppendToContainer_TcVnVector4_INT

	{attribute 'TcIecLibraryType'}
	{attribute 'external_name' := 'F_VN_AppendToContainer_TcVnVector4_INT_GUID_748F67D3_8551_39A4_3FC6_881669166664'}
	(* Append a single element of type TcVnVector4_INT to a container. *)
	FUNCTION F_VN_AppendToContainer_TcVnVector4_INT : HRESULT
	VAR_INPUT
		aElement	:	REFERENCE TO TcVnVector4_INT;	(* Single element to append to ipContainer *)
		ipContainer	:	ITcVnContainer;	(* Container to which the element will be appended *)
		hrPrev	:	HRESULT;	(* HRESULT indicating the result of previous operations (If SUCCEEDED(hrPrev) equals false, no operation is executed.) *)
	END_VAR

END_FUNCTION

// Functions/Basic Container Operations/F_VN_AppendToContainer/F_VN_AppendToContainer_TcVnVector4_LREAL

	{attribute 'TcIecLibraryType'}
	{attribute 'external_name' := 'F_VN_AppendToContainer_TcVnVector4_LREAL_GUID_1FB04494_25BC_3A6F_317E_B1721BC87D28'}
	(* Append a single element of type TcVnVector4_LREAL to a container. *)
	FUNCTION F_VN_AppendToContainer_TcVnVector4_LREAL : HRESULT
	VAR_INPUT
		aElement	:	REFERENCE TO TcVnVector4_LREAL;	(* Single element to append to ipContainer *)
		ipContainer	:	ITcVnContainer;	(* Container to which the element will be appended *)
		hrPrev	:	HRESULT;	(* HRESULT indicating the result of previous operations (If SUCCEEDED(hrPrev) equals false, no operation is executed.) *)
	END_VAR

END_FUNCTION

// Functions/Basic Container Operations/F_VN_AppendToContainer/F_VN_AppendToContainer_TcVnVector4_SINT

	{attribute 'TcIecLibraryType'}
	{attribute 'external_name' := 'F_VN_AppendToContainer_TcVnVector4_SINT_GUID_F864523C_2C39_358A_353C_C052C8CC0C37'}
	(* Append a single element of type TcVnVector4_SINT to a container. *)
	FUNCTION F_VN_AppendToContainer_TcVnVector4_SINT : HRESULT
	VAR_INPUT
		aElement	:	REFERENCE TO TcVnVector4_SINT;	(* Single element to append to ipContainer *)
		ipContainer	:	ITcVnContainer;	(* Container to which the element will be appended *)
		hrPrev	:	HRESULT;	(* HRESULT indicating the result of previous operations (If SUCCEEDED(hrPrev) equals false, no operation is executed.) *)
	END_VAR

END_FUNCTION

// Functions/Basic Container Operations/F_VN_AppendToContainer/F_VN_AppendToContainer_TcVnVector4_UINT

	{attribute 'TcIecLibraryType'}
	{attribute 'external_name' := 'F_VN_AppendToContainer_TcVnVector4_UINT_GUID_F413B457_2D7B_3278_0C44_D59DDCC999A6'}
	(* Append a single element of type TcVnVector4_UINT to a container. *)
	FUNCTION F_VN_AppendToContainer_TcVnVector4_UINT : HRESULT
	VAR_INPUT
		aElement	:	REFERENCE TO TcVnVector4_UINT;	(* Single element to append to ipContainer *)
		ipContainer	:	ITcVnContainer;	(* Container to which the element will be appended *)
		hrPrev	:	HRESULT;	(* HRESULT indicating the result of previous operations (If SUCCEEDED(hrPrev) equals false, no operation is executed.) *)
	END_VAR

END_FUNCTION

// Functions/Basic Container Operations/F_VN_AppendToContainer/F_VN_AppendToContainer_TcVnVector4_USINT

	{attribute 'TcIecLibraryType'}
	{attribute 'external_name' := 'F_VN_AppendToContainer_TcVnVector4_USINT_GUID_182A783A_C915_3F3B_1BC2_3A31A9190358'}
	(* Append a single element of type TcVnVector4_USINT to a container. *)
	FUNCTION F_VN_AppendToContainer_TcVnVector4_USINT : HRESULT
	VAR_INPUT
		aElement	:	REFERENCE TO TcVnVector4_USINT;	(* Single element to append to ipContainer *)
		ipContainer	:	ITcVnContainer;	(* Container to which the element will be appended *)
		hrPrev	:	HRESULT;	(* HRESULT indicating the result of previous operations (If SUCCEEDED(hrPrev) equals false, no operation is executed.) *)
	END_VAR

END_FUNCTION

// Functions/Basic Container Operations/F_VN_AppendToContainer/F_VN_AppendToContainer_UDINT

	{attribute 'TcIecLibraryType'}
	{attribute 'external_name' := 'F_VN_AppendToContainer_UDINT_GUID_F3DD6CFD_30E7_30B1_0148_5A567E71BF54'}
	(* Append a single element of type UDINT to a container. *)
	FUNCTION F_VN_AppendToContainer_UDINT : HRESULT
	VAR_INPUT
		nElement	:	UDINT;	(* Single element to append to ipContainer *)
		ipContainer	:	ITcVnContainer;	(* Container to which the element will be appended *)
		hrPrev	:	HRESULT;	(* HRESULT indicating the result of previous operations (If SUCCEEDED(hrPrev) equals false, no operation is executed.) *)
	END_VAR

END_FUNCTION

// Functions/Basic Container Operations/F_VN_AppendToContainer/F_VN_AppendToContainer_UINT

	{attribute 'TcIecLibraryType'}
	{attribute 'external_name' := 'F_VN_AppendToContainer_UINT_GUID_49962E15_7B80_3754_37EA_020A7E468E3A'}
	(* Append a single element of type UINT to a container. *)
	FUNCTION F_VN_AppendToContainer_UINT : HRESULT
	VAR_INPUT
		nElement	:	UINT;	(* Single element to append to ipContainer *)
		ipContainer	:	ITcVnContainer;	(* Container to which the element will be appended *)
		hrPrev	:	HRESULT;	(* HRESULT indicating the result of previous operations (If SUCCEEDED(hrPrev) equals false, no operation is executed.) *)
	END_VAR

END_FUNCTION

// Functions/Basic Container Operations/F_VN_AppendToContainer/F_VN_AppendToContainer_ULINT

	{attribute 'TcIecLibraryType'}
	{attribute 'external_name' := 'F_VN_AppendToContainer_ULINT_GUID_C58B30C6_57F1_341F_34C5_57833E30BC09'}
	(* Append a single element of type ULINT to a container. *)
	FUNCTION F_VN_AppendToContainer_ULINT : HRESULT
	VAR_INPUT
		nElement	:	ULINT;	(* Single element to append to ipContainer *)
		ipContainer	:	ITcVnContainer;	(* Container to which the element will be appended *)
		hrPrev	:	HRESULT;	(* HRESULT indicating the result of previous operations (If SUCCEEDED(hrPrev) equals false, no operation is executed.) *)
	END_VAR

END_FUNCTION

// Functions/Basic Container Operations/F_VN_AppendToContainer/F_VN_AppendToContainer_USINT

	{attribute 'TcIecLibraryType'}
	{attribute 'external_name' := 'F_VN_AppendToContainer_USINT_GUID_7B0C1157_B274_3307_2BAD_88003EAB0B7C'}
	(* Append a single element of type USINT to a container. *)
	FUNCTION F_VN_AppendToContainer_USINT : HRESULT
	VAR_INPUT
		nElement	:	USINT;	(* Single element to append to ipContainer *)
		ipContainer	:	ITcVnContainer;	(* Container to which the element will be appended *)
		hrPrev	:	HRESULT;	(* HRESULT indicating the result of previous operations (If SUCCEEDED(hrPrev) equals false, no operation is executed.) *)
	END_VAR

END_FUNCTION

// Functions/Basic Container Operations/F_VN_FillContainer/F_VN_FillContainer_DINT

	{attribute 'TcIecLibraryType'}
	{attribute 'external_name' := 'F_VN_FillContainer_DINT_GUID_7F931FAA_62FC_3633_201C_432C8F9E5852'}
	(* Fill the container with the specified value. Only possible for containers with basic elements. *)
	FUNCTION F_VN_FillContainer_DINT : HRESULT
	VAR_INPUT
		ipContainer	:	ITcVnContainer;	(* Container with basic elements *)
		nValue	:	DINT;	(* Value to set the container elements *)
		hrPrev	:	HRESULT;	(* HRESULT indicating the result of previous operations (If SUCCEEDED(hrPrev) equals false, no operation is executed.) *)
	END_VAR

END_FUNCTION

// Functions/Basic Container Operations/F_VN_FillContainer/F_VN_FillContainer_INT

	{attribute 'TcIecLibraryType'}
	{attribute 'external_name' := 'F_VN_FillContainer_INT_GUID_F97E92AB_9CB6_3350_3960_66DD53C6B1AD'}
	(* Fill the container with the specified value. Only possible for containers with basic elements. *)
	FUNCTION F_VN_FillContainer_INT : HRESULT
	VAR_INPUT
		ipContainer	:	ITcVnContainer;	(* Container with basic elements *)
		nValue	:	INT;	(* Value to set the container elements *)
		hrPrev	:	HRESULT;	(* HRESULT indicating the result of previous operations (If SUCCEEDED(hrPrev) equals false, no operation is executed.) *)
	END_VAR

END_FUNCTION

// Functions/Basic Container Operations/F_VN_FillContainer/F_VN_FillContainer_LREAL

	{attribute 'TcIecLibraryType'}
	{attribute 'external_name' := 'F_VN_FillContainer_LREAL_GUID_FA92836B_9461_39ED_21BF_3EA64F68BF45'}
	(* Fill the container with the specified value. Only possible for containers with basic elements. *)
	FUNCTION F_VN_FillContainer_LREAL : HRESULT
	VAR_INPUT
		ipContainer	:	ITcVnContainer;	(* Container with basic elements *)
		fValue	:	LREAL;	(* Value to set the container elements *)
		hrPrev	:	HRESULT;	(* HRESULT indicating the result of previous operations (If SUCCEEDED(hrPrev) equals false, no operation is executed.) *)
	END_VAR

END_FUNCTION

// Functions/Basic Container Operations/F_VN_FillContainer/F_VN_FillContainer_REAL

	{attribute 'TcIecLibraryType'}
	{attribute 'external_name' := 'F_VN_FillContainer_REAL_GUID_A798AD39_8D46_3334_1F07_ADC7ECA2767F'}
	(* Fill the container with the specified value. Only possible for containers with basic elements. *)
	FUNCTION F_VN_FillContainer_REAL : HRESULT
	VAR_INPUT
		ipContainer	:	ITcVnContainer;	(* Container with basic elements *)
		fValue	:	REAL;	(* Value to set the container elements *)
		hrPrev	:	HRESULT;	(* HRESULT indicating the result of previous operations (If SUCCEEDED(hrPrev) equals false, no operation is executed.) *)
	END_VAR

END_FUNCTION

// Functions/Basic Container Operations/F_VN_FillContainer/F_VN_FillContainer_SINT

	{attribute 'TcIecLibraryType'}
	{attribute 'external_name' := 'F_VN_FillContainer_SINT_GUID_80A4EA2E_FAA5_3110_2D88_9E788EE88C4A'}
	(* Fill the container with the specified value. Only possible for containers with basic elements. *)
	FUNCTION F_VN_FillContainer_SINT : HRESULT
	VAR_INPUT
		ipContainer	:	ITcVnContainer;	(* Container with basic elements *)
		nValue	:	SINT;	(* Value to set the container elements *)
		hrPrev	:	HRESULT;	(* HRESULT indicating the result of previous operations (If SUCCEEDED(hrPrev) equals false, no operation is executed.) *)
	END_VAR

END_FUNCTION

// Functions/Basic Container Operations/F_VN_FillContainer/F_VN_FillContainer_TcVnDMatch

	{attribute 'TcIecLibraryType'}
	{attribute 'external_name' := 'F_VN_FillContainer_TcVnDMatch_GUID_ED645E1C_85A6_3546_2AAD_5FB9B394FE82'}
	(* Fill the container with the specified value. Only possible for containers with basic elements. *)
	FUNCTION F_VN_FillContainer_TcVnDMatch : HRESULT
	VAR_INPUT
		ipContainer	:	ITcVnContainer;	(* Container with basic elements *)
		stValue	:	REFERENCE TO TcVnDMatch;	(* Value to set the container elements *)
		hrPrev	:	HRESULT;	(* HRESULT indicating the result of previous operations (If SUCCEEDED(hrPrev) equals false, no operation is executed.) *)
	END_VAR

END_FUNCTION

// Functions/Basic Container Operations/F_VN_FillContainer/F_VN_FillContainer_TcVnKeyPoint

	{attribute 'TcIecLibraryType'}
	{attribute 'external_name' := 'F_VN_FillContainer_TcVnKeyPoint_GUID_67D41008_FB29_3015_234C_3406A002A695'}
	(* Fill the container with the specified value. Only possible for containers with basic elements. *)
	FUNCTION F_VN_FillContainer_TcVnKeyPoint : HRESULT
	VAR_INPUT
		ipContainer	:	ITcVnContainer;	(* Container with basic elements *)
		stValue	:	REFERENCE TO TcVnKeyPoint;	(* Value to set the container elements *)
		hrPrev	:	HRESULT;	(* HRESULT indicating the result of previous operations (If SUCCEEDED(hrPrev) equals false, no operation is executed.) *)
	END_VAR

END_FUNCTION

// Functions/Basic Container Operations/F_VN_FillContainer/F_VN_FillContainer_TcVnPoint2_DINT

	{attribute 'TcIecLibraryType'}
	{attribute 'external_name' := 'F_VN_FillContainer_TcVnPoint2_DINT_GUID_7D4BDF54_0732_3865_2C81_9624658CC974'}
	(* Fill the container with the specified value. Only possible for containers with basic elements. *)
	FUNCTION F_VN_FillContainer_TcVnPoint2_DINT : HRESULT
	VAR_INPUT
		ipContainer	:	ITcVnContainer;	(* Container with basic elements *)
		aValue	:	REFERENCE TO TcVnPoint2_DINT;	(* Value to set the container elements *)
		hrPrev	:	HRESULT;	(* HRESULT indicating the result of previous operations (If SUCCEEDED(hrPrev) equals false, no operation is executed.) *)
	END_VAR

END_FUNCTION

// Functions/Basic Container Operations/F_VN_FillContainer/F_VN_FillContainer_TcVnPoint2_LREAL

	{attribute 'TcIecLibraryType'}
	{attribute 'external_name' := 'F_VN_FillContainer_TcVnPoint2_LREAL_GUID_DD962A39_D926_3E09_0537_4D7162C961B6'}
	(* Fill the container with the specified value. Only possible for containers with basic elements. *)
	FUNCTION F_VN_FillContainer_TcVnPoint2_LREAL : HRESULT
	VAR_INPUT
		ipContainer	:	ITcVnContainer;	(* Container with basic elements *)
		aValue	:	REFERENCE TO TcVnPoint2_LREAL;	(* Value to set the container elements *)
		hrPrev	:	HRESULT;	(* HRESULT indicating the result of previous operations (If SUCCEEDED(hrPrev) equals false, no operation is executed.) *)
	END_VAR

END_FUNCTION

// Functions/Basic Container Operations/F_VN_FillContainer/F_VN_FillContainer_TcVnPoint2_REAL

	{attribute 'TcIecLibraryType'}
	{attribute 'external_name' := 'F_VN_FillContainer_TcVnPoint2_REAL_GUID_72279693_0711_34CB_2AD3_26F22DB58685'}
	(* Fill the container with the specified value. Only possible for containers with basic elements. *)
	FUNCTION F_VN_FillContainer_TcVnPoint2_REAL : HRESULT
	VAR_INPUT
		ipContainer	:	ITcVnContainer;	(* Container with basic elements *)
		aValue	:	REFERENCE TO TcVnPoint2_REAL;	(* Value to set the container elements *)
		hrPrev	:	HRESULT;	(* HRESULT indicating the result of previous operations (If SUCCEEDED(hrPrev) equals false, no operation is executed.) *)
	END_VAR

END_FUNCTION

// Functions/Basic Container Operations/F_VN_FillContainer/F_VN_FillContainer_TcVnPoint3_LREAL

	{attribute 'TcIecLibraryType'}
	{attribute 'external_name' := 'F_VN_FillContainer_TcVnPoint3_LREAL_GUID_8967D304_0054_30BE_1C00_039388504133'}
	(* Fill the container with the specified value. Only possible for containers with basic elements. *)
	FUNCTION F_VN_FillContainer_TcVnPoint3_LREAL : HRESULT
	VAR_INPUT
		ipContainer	:	ITcVnContainer;	(* Container with basic elements *)
		aValue	:	REFERENCE TO TcVnPoint3_LREAL;	(* Value to set the container elements *)
		hrPrev	:	HRESULT;	(* HRESULT indicating the result of previous operations (If SUCCEEDED(hrPrev) equals false, no operation is executed.) *)
	END_VAR

END_FUNCTION

// Functions/Basic Container Operations/F_VN_FillContainer/F_VN_FillContainer_TcVnPoint3_REAL

	{attribute 'TcIecLibraryType'}
	{attribute 'external_name' := 'F_VN_FillContainer_TcVnPoint3_REAL_GUID_68EE3077_6FEB_3104_26AE_1AB52F23CC70'}
	(* Fill the container with the specified value. Only possible for containers with basic elements. *)
	FUNCTION F_VN_FillContainer_TcVnPoint3_REAL : HRESULT
	VAR_INPUT
		ipContainer	:	ITcVnContainer;	(* Container with basic elements *)
		aValue	:	REFERENCE TO TcVnPoint3_REAL;	(* Value to set the container elements *)
		hrPrev	:	HRESULT;	(* HRESULT indicating the result of previous operations (If SUCCEEDED(hrPrev) equals false, no operation is executed.) *)
	END_VAR

END_FUNCTION

// Functions/Basic Container Operations/F_VN_FillContainer/F_VN_FillContainer_TcVnRectangle_DINT

	{attribute 'TcIecLibraryType'}
	{attribute 'external_name' := 'F_VN_FillContainer_TcVnRectangle_DINT_GUID_1827139B_269C_3DF5_02B1_3D9AFDDE8A96'}
	(* Fill the container with the specified value. Only possible for containers with basic elements. *)
	FUNCTION F_VN_FillContainer_TcVnRectangle_DINT : HRESULT
	VAR_INPUT
		ipContainer	:	ITcVnContainer;	(* Container with basic elements *)
		stValue	:	REFERENCE TO TcVnRectangle_DINT;	(* Value to set the container elements *)
		hrPrev	:	HRESULT;	(* HRESULT indicating the result of previous operations (If SUCCEEDED(hrPrev) equals false, no operation is executed.) *)
	END_VAR

END_FUNCTION

// Functions/Basic Container Operations/F_VN_FillContainer/F_VN_FillContainer_TcVnVector2_DINT

	{attribute 'TcIecLibraryType'}
	{attribute 'external_name' := 'F_VN_FillContainer_TcVnVector2_DINT_GUID_22B31A28_8A47_378F_0589_59D7E89F162D'}
	(* Fill the container with the specified value. Only possible for containers with basic elements. *)
	FUNCTION F_VN_FillContainer_TcVnVector2_DINT : HRESULT
	VAR_INPUT
		ipContainer	:	ITcVnContainer;	(* Container with basic elements *)
		aValue	:	REFERENCE TO TcVnVector2_DINT;	(* Value to set the container elements *)
		hrPrev	:	HRESULT;	(* HRESULT indicating the result of previous operations (If SUCCEEDED(hrPrev) equals false, no operation is executed.) *)
	END_VAR

END_FUNCTION

// Functions/Basic Container Operations/F_VN_FillContainer/F_VN_FillContainer_TcVnVector2_INT

	{attribute 'TcIecLibraryType'}
	{attribute 'external_name' := 'F_VN_FillContainer_TcVnVector2_INT_GUID_F21369A5_3216_3A3B_339E_49660A943AD3'}
	(* Fill the container with the specified value. Only possible for containers with basic elements. *)
	FUNCTION F_VN_FillContainer_TcVnVector2_INT : HRESULT
	VAR_INPUT
		ipContainer	:	ITcVnContainer;	(* Container with basic elements *)
		aValue	:	REFERENCE TO TcVnVector2_INT;	(* Value to set the container elements *)
		hrPrev	:	HRESULT;	(* HRESULT indicating the result of previous operations (If SUCCEEDED(hrPrev) equals false, no operation is executed.) *)
	END_VAR

END_FUNCTION

// Functions/Basic Container Operations/F_VN_FillContainer/F_VN_FillContainer_TcVnVector2_REAL

	{attribute 'TcIecLibraryType'}
	{attribute 'external_name' := 'F_VN_FillContainer_TcVnVector2_REAL_GUID_B5727D3A_9409_3930_3683_A68FE7F31C49'}
	(* Fill the container with the specified value. Only possible for containers with basic elements. *)
	FUNCTION F_VN_FillContainer_TcVnVector2_REAL : HRESULT
	VAR_INPUT
		ipContainer	:	ITcVnContainer;	(* Container with basic elements *)
		aValue	:	REFERENCE TO TcVnVector2_REAL;	(* Value to set the container elements *)
		hrPrev	:	HRESULT;	(* HRESULT indicating the result of previous operations (If SUCCEEDED(hrPrev) equals false, no operation is executed.) *)
	END_VAR

END_FUNCTION

// Functions/Basic Container Operations/F_VN_FillContainer/F_VN_FillContainer_TcVnVector2_SINT

	{attribute 'TcIecLibraryType'}
	{attribute 'external_name' := 'F_VN_FillContainer_TcVnVector2_SINT_GUID_02F3DCAE_780D_3605_2208_50CC7B9B1CA1'}
	(* Fill the container with the specified value. Only possible for containers with basic elements. *)
	FUNCTION F_VN_FillContainer_TcVnVector2_SINT : HRESULT
	VAR_INPUT
		ipContainer	:	ITcVnContainer;	(* Container with basic elements *)
		aValue	:	REFERENCE TO TcVnVector2_SINT;	(* Value to set the container elements *)
		hrPrev	:	HRESULT;	(* HRESULT indicating the result of previous operations (If SUCCEEDED(hrPrev) equals false, no operation is executed.) *)
	END_VAR

END_FUNCTION

// Functions/Basic Container Operations/F_VN_FillContainer/F_VN_FillContainer_TcVnVector2_UINT

	{attribute 'TcIecLibraryType'}
	{attribute 'external_name' := 'F_VN_FillContainer_TcVnVector2_UINT_GUID_82ED187A_35E1_3DF3_18D0_D71F8378DF9C'}
	(* Fill the container with the specified value. Only possible for containers with basic elements. *)
	FUNCTION F_VN_FillContainer_TcVnVector2_UINT : HRESULT
	VAR_INPUT
		ipContainer	:	ITcVnContainer;	(* Container with basic elements *)
		aValue	:	REFERENCE TO TcVnVector2_UINT;	(* Value to set the container elements *)
		hrPrev	:	HRESULT;	(* HRESULT indicating the result of previous operations (If SUCCEEDED(hrPrev) equals false, no operation is executed.) *)
	END_VAR

END_FUNCTION

// Functions/Basic Container Operations/F_VN_FillContainer/F_VN_FillContainer_TcVnVector2_USINT

	{attribute 'TcIecLibraryType'}
	{attribute 'external_name' := 'F_VN_FillContainer_TcVnVector2_USINT_GUID_AA2DD3AD_A90B_335A_1E6C_1F3290ED816C'}
	(* Fill the container with the specified value. Only possible for containers with basic elements. *)
	FUNCTION F_VN_FillContainer_TcVnVector2_USINT : HRESULT
	VAR_INPUT
		ipContainer	:	ITcVnContainer;	(* Container with basic elements *)
		aValue	:	REFERENCE TO TcVnVector2_USINT;	(* Value to set the container elements *)
		hrPrev	:	HRESULT;	(* HRESULT indicating the result of previous operations (If SUCCEEDED(hrPrev) equals false, no operation is executed.) *)
	END_VAR

END_FUNCTION

// Functions/Basic Container Operations/F_VN_FillContainer/F_VN_FillContainer_TcVnVector3_INT

	{attribute 'TcIecLibraryType'}
	{attribute 'external_name' := 'F_VN_FillContainer_TcVnVector3_INT_GUID_69ED6B74_EB53_3343_3041_1DCE93887E2B'}
	(* Fill the container with the specified value. Only possible for containers with basic elements. *)
	FUNCTION F_VN_FillContainer_TcVnVector3_INT : HRESULT
	VAR_INPUT
		ipContainer	:	ITcVnContainer;	(* Container with basic elements *)
		aValue	:	REFERENCE TO TcVnVector3_INT;	(* Value to set the container elements *)
		hrPrev	:	HRESULT;	(* HRESULT indicating the result of previous operations (If SUCCEEDED(hrPrev) equals false, no operation is executed.) *)
	END_VAR

END_FUNCTION

// Functions/Basic Container Operations/F_VN_FillContainer/F_VN_FillContainer_TcVnVector3_REAL

	{attribute 'TcIecLibraryType'}
	{attribute 'external_name' := 'F_VN_FillContainer_TcVnVector3_REAL_GUID_EC94386E_E0D5_30C6_087A_0B5E2A0067FF'}
	(* Fill the container with the specified value. Only possible for containers with basic elements. *)
	FUNCTION F_VN_FillContainer_TcVnVector3_REAL : HRESULT
	VAR_INPUT
		ipContainer	:	ITcVnContainer;	(* Container with basic elements *)
		aValue	:	REFERENCE TO TcVnVector3_REAL;	(* Value to set the container elements *)
		hrPrev	:	HRESULT;	(* HRESULT indicating the result of previous operations (If SUCCEEDED(hrPrev) equals false, no operation is executed.) *)
	END_VAR

END_FUNCTION

// Functions/Basic Container Operations/F_VN_FillContainer/F_VN_FillContainer_TcVnVector3_SINT

	{attribute 'TcIecLibraryType'}
	{attribute 'external_name' := 'F_VN_FillContainer_TcVnVector3_SINT_GUID_05ACDA77_39B7_3BA4_1290_3CCCF530D331'}
	(* Fill the container with the specified value. Only possible for containers with basic elements. *)
	FUNCTION F_VN_FillContainer_TcVnVector3_SINT : HRESULT
	VAR_INPUT
		ipContainer	:	ITcVnContainer;	(* Container with basic elements *)
		aValue	:	REFERENCE TO TcVnVector3_SINT;	(* Value to set the container elements *)
		hrPrev	:	HRESULT;	(* HRESULT indicating the result of previous operations (If SUCCEEDED(hrPrev) equals false, no operation is executed.) *)
	END_VAR

END_FUNCTION

// Functions/Basic Container Operations/F_VN_FillContainer/F_VN_FillContainer_TcVnVector3_UINT

	{attribute 'TcIecLibraryType'}
	{attribute 'external_name' := 'F_VN_FillContainer_TcVnVector3_UINT_GUID_3CC3C3DB_0C1E_3F9F_29FA_B5A6DF495AF3'}
	(* Fill the container with the specified value. Only possible for containers with basic elements. *)
	FUNCTION F_VN_FillContainer_TcVnVector3_UINT : HRESULT
	VAR_INPUT
		ipContainer	:	ITcVnContainer;	(* Container with basic elements *)
		aValue	:	REFERENCE TO TcVnVector3_UINT;	(* Value to set the container elements *)
		hrPrev	:	HRESULT;	(* HRESULT indicating the result of previous operations (If SUCCEEDED(hrPrev) equals false, no operation is executed.) *)
	END_VAR

END_FUNCTION

// Functions/Basic Container Operations/F_VN_FillContainer/F_VN_FillContainer_TcVnVector3_USINT

	{attribute 'TcIecLibraryType'}
	{attribute 'external_name' := 'F_VN_FillContainer_TcVnVector3_USINT_GUID_5B5D84DF_3033_3DE9_1003_84C98E45743E'}
	(* Fill the container with the specified value. Only possible for containers with basic elements. *)
	FUNCTION F_VN_FillContainer_TcVnVector3_USINT : HRESULT
	VAR_INPUT
		ipContainer	:	ITcVnContainer;	(* Container with basic elements *)
		aValue	:	REFERENCE TO TcVnVector3_USINT;	(* Value to set the container elements *)
		hrPrev	:	HRESULT;	(* HRESULT indicating the result of previous operations (If SUCCEEDED(hrPrev) equals false, no operation is executed.) *)
	END_VAR

END_FUNCTION

// Functions/Basic Container Operations/F_VN_FillContainer/F_VN_FillContainer_TcVnVector4_DINT

	{attribute 'TcIecLibraryType'}
	{attribute 'external_name' := 'F_VN_FillContainer_TcVnVector4_DINT_GUID_E3B5AD4D_5D00_37E6_2E28_39259777A710'}
	(* Fill the container with the specified value. Only possible for containers with basic elements. *)
	FUNCTION F_VN_FillContainer_TcVnVector4_DINT : HRESULT
	VAR_INPUT
		ipContainer	:	ITcVnContainer;	(* Container with basic elements *)
		aValue	:	REFERENCE TO TcVnVector4_DINT;	(* Value to set the container elements *)
		hrPrev	:	HRESULT;	(* HRESULT indicating the result of previous operations (If SUCCEEDED(hrPrev) equals false, no operation is executed.) *)
	END_VAR

END_FUNCTION

// Functions/Basic Container Operations/F_VN_FillContainer/F_VN_FillContainer_TcVnVector4_INT

	{attribute 'TcIecLibraryType'}
	{attribute 'external_name' := 'F_VN_FillContainer_TcVnVector4_INT_GUID_3D043214_AE9C_300E_3F1A_02B8BD32C693'}
	(* Fill the container with the specified value. Only possible for containers with basic elements. *)
	FUNCTION F_VN_FillContainer_TcVnVector4_INT : HRESULT
	VAR_INPUT
		ipContainer	:	ITcVnContainer;	(* Container with basic elements *)
		aValue	:	REFERENCE TO TcVnVector4_INT;	(* Value to set the container elements *)
		hrPrev	:	HRESULT;	(* HRESULT indicating the result of previous operations (If SUCCEEDED(hrPrev) equals false, no operation is executed.) *)
	END_VAR

END_FUNCTION

// Functions/Basic Container Operations/F_VN_FillContainer/F_VN_FillContainer_TcVnVector4_LREAL

	{attribute 'TcIecLibraryType'}
	{attribute 'external_name' := 'F_VN_FillContainer_TcVnVector4_LREAL_GUID_3A3537BF_F86F_3EDD_1DE5_63FB125E5374'}
	(* Fill the container with the specified value. Only possible for containers with basic elements. *)
	FUNCTION F_VN_FillContainer_TcVnVector4_LREAL : HRESULT
	VAR_INPUT
		ipContainer	:	ITcVnContainer;	(* Container with basic elements *)
		aValue	:	REFERENCE TO TcVnVector4_LREAL;	(* Value to set the container elements *)
		hrPrev	:	HRESULT;	(* HRESULT indicating the result of previous operations (If SUCCEEDED(hrPrev) equals false, no operation is executed.) *)
	END_VAR

END_FUNCTION

// Functions/Basic Container Operations/F_VN_FillContainer/F_VN_FillContainer_TcVnVector4_SINT

	{attribute 'TcIecLibraryType'}
	{attribute 'external_name' := 'F_VN_FillContainer_TcVnVector4_SINT_GUID_C9C700F1_62C0_33A1_38B5_3540B3CACEA3'}
	(* Fill the container with the specified value. Only possible for containers with basic elements. *)
	FUNCTION F_VN_FillContainer_TcVnVector4_SINT : HRESULT
	VAR_INPUT
		ipContainer	:	ITcVnContainer;	(* Container with basic elements *)
		aValue	:	REFERENCE TO TcVnVector4_SINT;	(* Value to set the container elements *)
		hrPrev	:	HRESULT;	(* HRESULT indicating the result of previous operations (If SUCCEEDED(hrPrev) equals false, no operation is executed.) *)
	END_VAR

END_FUNCTION

// Functions/Basic Container Operations/F_VN_FillContainer/F_VN_FillContainer_TcVnVector4_UINT

	{attribute 'TcIecLibraryType'}
	{attribute 'external_name' := 'F_VN_FillContainer_TcVnVector4_UINT_GUID_04F78A70_ED82_371B_0E13_F31528232EE8'}
	(* Fill the container with the specified value. Only possible for containers with basic elements. *)
	FUNCTION F_VN_FillContainer_TcVnVector4_UINT : HRESULT
	VAR_INPUT
		ipContainer	:	ITcVnContainer;	(* Container with basic elements *)
		aValue	:	REFERENCE TO TcVnVector4_UINT;	(* Value to set the container elements *)
		hrPrev	:	HRESULT;	(* HRESULT indicating the result of previous operations (If SUCCEEDED(hrPrev) equals false, no operation is executed.) *)
	END_VAR

END_FUNCTION

// Functions/Basic Container Operations/F_VN_FillContainer/F_VN_FillContainer_TcVnVector4_USINT

	{attribute 'TcIecLibraryType'}
	{attribute 'external_name' := 'F_VN_FillContainer_TcVnVector4_USINT_GUID_D509B950_76E5_3370_254C_01A5F083CCB4'}
	(* Fill the container with the specified value. Only possible for containers with basic elements. *)
	FUNCTION F_VN_FillContainer_TcVnVector4_USINT : HRESULT
	VAR_INPUT
		ipContainer	:	ITcVnContainer;	(* Container with basic elements *)
		aValue	:	REFERENCE TO TcVnVector4_USINT;	(* Value to set the container elements *)
		hrPrev	:	HRESULT;	(* HRESULT indicating the result of previous operations (If SUCCEEDED(hrPrev) equals false, no operation is executed.) *)
	END_VAR

END_FUNCTION

// Functions/Basic Container Operations/F_VN_FillContainer/F_VN_FillContainer_UDINT

	{attribute 'TcIecLibraryType'}
	{attribute 'external_name' := 'F_VN_FillContainer_UDINT_GUID_543AE012_51AF_377D_04C8_92427A066FD5'}
	(* Fill the container with the specified value. Only possible for containers with basic elements. *)
	FUNCTION F_VN_FillContainer_UDINT : HRESULT
	VAR_INPUT
		ipContainer	:	ITcVnContainer;	(* Container with basic elements *)
		nValue	:	UDINT;	(* Value to set the container elements *)
		hrPrev	:	HRESULT;	(* HRESULT indicating the result of previous operations (If SUCCEEDED(hrPrev) equals false, no operation is executed.) *)
	END_VAR

END_FUNCTION

// Functions/Basic Container Operations/F_VN_FillContainer/F_VN_FillContainer_UINT

	{attribute 'TcIecLibraryType'}
	{attribute 'external_name' := 'F_VN_FillContainer_UINT_GUID_C26554B6_307E_38ED_1B49_E6D9DA3E08D6'}
	(* Fill the container with the specified value. Only possible for containers with basic elements. *)
	FUNCTION F_VN_FillContainer_UINT : HRESULT
	VAR_INPUT
		ipContainer	:	ITcVnContainer;	(* Container with basic elements *)
		nValue	:	UINT;	(* Value to set the container elements *)
		hrPrev	:	HRESULT;	(* HRESULT indicating the result of previous operations (If SUCCEEDED(hrPrev) equals false, no operation is executed.) *)
	END_VAR

END_FUNCTION

// Functions/Basic Container Operations/F_VN_FillContainer/F_VN_FillContainer_ULINT

	{attribute 'TcIecLibraryType'}
	{attribute 'external_name' := 'F_VN_FillContainer_ULINT_GUID_69B2762F_8D6C_349C_205F_B49F0991C3B5'}
	(* Fill the container with the specified value. Only possible for containers with basic elements. *)
	FUNCTION F_VN_FillContainer_ULINT : HRESULT
	VAR_INPUT
		ipContainer	:	ITcVnContainer;	(* Container with basic elements *)
		nValue	:	ULINT;	(* Value to set the container elements *)
		hrPrev	:	HRESULT;	(* HRESULT indicating the result of previous operations (If SUCCEEDED(hrPrev) equals false, no operation is executed.) *)
	END_VAR

END_FUNCTION

// Functions/Basic Container Operations/F_VN_FillContainer/F_VN_FillContainer_USINT

	{attribute 'TcIecLibraryType'}
	{attribute 'external_name' := 'F_VN_FillContainer_USINT_GUID_03424834_14D2_31C3_2C73_CE9ACFE9DAE7'}
	(* Fill the container with the specified value. Only possible for containers with basic elements. *)
	FUNCTION F_VN_FillContainer_USINT : HRESULT
	VAR_INPUT
		ipContainer	:	ITcVnContainer;	(* Container with basic elements *)
		nValue	:	USINT;	(* Value to set the container elements *)
		hrPrev	:	HRESULT;	(* HRESULT indicating the result of previous operations (If SUCCEEDED(hrPrev) equals false, no operation is executed.) *)
	END_VAR

END_FUNCTION

// Functions/Basic Container Operations/F_VN_FillContainerExp/F_VN_FillContainerExp_DINT

